C03633=1108.269,417.055,404.541,-178.654,16.489,151.227
C03634=1108.274,417.302,404.502,-178.652,16.496,151.228
C03635=1108.279,417.549,404.464,-178.650,16.503,151.230
C03636=1108.285,417.796,404.425,-178.649,16.510,151.231
C03637=1108.291,418.042,404.386,-178.647,16.517,151.232
C03638=1108.297,418.289,404.346,-178.645,16.524,151.234
C03639=1108.302,418.536,404.307,-178.644,16.531,151.235
C03640=1108.307,418.783,404.267,-178.642,16.538,151.237
C03641=1108.313,419.030,404.228,-178.640,16.545,151.238
C03642=1108.319,419.276,404.189,-178.639,16.553,151.240
C03643=1108.325,419.523,404.149,-178.638,16.560,151.241
C03644=1108.330,419.770,404.110,-178.636,16.567,151.243
C03645=1108.336,420.017,404.071,-178.634,16.574,151.244
C03646=1108.342,420.264,404.033,-178.632,16.582,151.246
C03647=1108.347,420.510,403.992,-178.631,16.589,151.247
C03648=1108.353,420.757,403.953,-178.629,16.596,151.249
C03649=1108.358,421.004,403.914,-178.627,16.603,151.250
C03650=1108.364,421.251,403.874,-178.626,16.611,151.252
C03651=1108.370,421.497,403.835,-178.625,16.618,151.254
C03652=1108.375,421.745,403.795,-178.623,16.625,151.255
C03653=1108.381,421.991,403.756,-178.621,16.633,151.257
C03654=1108.387,422.238,403.717,-178.619,16.640,151.258
C03655=1108.392,422.485,403.678,-178.618,16.648,151.260
C03656=1108.398,422.732,403.638,-178.616,16.655,151.261
C03657=1108.403,422.978,403.598,-178.615,16.663,151.263
C03658=1108.409,423.225,403.558,-178.614,16.670,151.265
C03659=1108.414,423.443,403.524,-178.612,16.678,151.266
C03660=1108.419,423.661,403.489,-178.611,16.684,151.268
C03661=1108.424,423.879,403.454,-178.610,16.691,151.269
C03662=1108.429,424.099,403.418,-178.608,16.698,151.271
C03663=1108.434,424.317,403.383,-178.607,16.704,151.272
C03664=1108.439,424.535,403.348,-178.606,16.712,151.274
C03665=1108.443,424.753,403.313,-178.604,16.718,151.275
C03666=1108.449,424.972,403.278,-178.603,16.725,151.277
C03667=1108.454,425.218,403.238,-178.602,16.733,151.278
C03668=1108.460,425.465,403.198,-178.600,16.741,151.280
C03669=1108.465,425.712,403.158,-178.599,16.749,151.282
C03670=1108.471,425.959,403.119,-178.598,16.757,151.283
C03671=1108.477,426.205,403.079,-178.596,16.764,151.285
C03672=1108.482,426.452,403.039,-178.595,16.773,151.287
C03673=1108.488,426.698,402.999,-178.593,16.781,151.289
C03674=1108.493,426.945,402.959,-178.592,16.789,151.290
C03675=1108.500,427.192,402.919,-178.591,16.797,151.292
C03676=1108.504,427.439,402.879,-178.589,16.805,151.294
C03677=1108.511,427.685,402.839,-178.588,16.813,151.296
C03678=1108.515,427.932,402.800,-178.587,16.821,151.298
C03679=1108.522,428.178,402.760,-178.585,16.829,151.299
C03680=1108.527,428.426,402.719,-178.584,16.837,151.301
C03681=1108.533,428.672,402.680,-178.583,16.845,151.303
C03682=1108.539,428.918,402.639,-178.582,16.854,151.305
C03683=1108.544,429.165,402.600,-178.580,16.862,151.307
C03684=1108.550,429.412,402.559,-178.579,16.870,151.309
C03685=1108.556,429.659,402.520,-178.578,16.879,151.311
C03686=1108.561,429.905,402.479,-178.577,16.887,151.312
C03687=1108.566,430.152,402.439,-178.575,16.896,151.314
C03688=1108.572,430.398,402.399,-178.574,16.904,151.316
C03689=1108.578,430.645,402.359,-178.573,16.913,151.318
C03690=1108.584,430.892,402.319,-178.572,16.921,151.320
C03691=1108.589,431.138,402.278,-178.571,16.930,151.322
C03692=1108.595,431.384,402.238,-178.570,16.938,151.324
C03693=1108.601,431.632,402.198,-178.568,16.946,151.326
C03694=1108.606,431.878,402.158,-178.567,16.956,151.328
C03695=1108.611,432.125,402.117,-178.566,16.964,151.330
C03696=1108.617,432.371,402.076,-178.565,16.973,151.332
C03697=1108.623,432.617,402.036,-178.564,16.981,151.334
C03698=1108.628,432.864,401.996,-178.563,16.990,151.336
C03699=1108.634,433.111,401.956,-178.561,16.999,151.338
C03700=1108.640,433.357,401.916,-178.560,17.008,151.340
C03701=1108.645,433.604,401.875,-178.560,17.017,151.342
C03702=1108.651,433.851,401.834,-178.559,17.025,151.344
C03703=1108.656,434.097,401.794,-178.558,17.034,151.346
C03704=1108.662,434.344,401.753,-178.556,17.044,151.348
C03705=1108.667,434.591,401.713,-178.556,17.052,151.351
C03706=1108.673,434.837,401.673,-178.555,17.061,151.353
C03707=1108.679,435.083,401.632,-178.553,17.071,151.355
C03708=1108.684,435.330,401.591,-178.553,17.080,151.357
C03709=1108.689,435.576,401.551,-178.552,17.089,151.359
C03710=1108.695,435.823,401.510,-178.551,17.098,151.361
C03711=1108.701,436.069,401.469,-178.550,17.107,151.364
C03712=1108.706,436.315,401.428,-178.549,17.117,151.366
C03713=1108.712,436.562,401.388,-178.549,17.126,151.368
C03714=1108.717,436.809,401.347,-178.547,17.135,151.370
C03715=1108.723,437.037,401.310,-178.546,17.144,151.372
C03716=1108.727,437.265,401.272,-178.545,17.153,151.374
C03717=1108.733,437.493,401.234,-178.545,17.161,151.376
C03718=1108.738,437.721,401.196,-178.545,17.170,151.379
C03719=1108.743,437.949,401.159,-178.544,17.179,151.381
C03720=1108.749,438.177,401.121,-178.543,17.188,151.383
C03721=1108.754,438.406,401.083,-178.542,17.196,151.385
C03722=1108.758,438.634,401.046,-178.541,17.205,151.387
C03723=1108.764,438.880,401.004,-178.541,17.215,151.389
C03724=1108.770,439.127,400.963,-178.540,17.224,151.392
C03725=1108.776,439.373,400.922,-178.539,17.234,151.394
C03726=1108.782,439.620,400.881,-178.538,17.244,151.396
C03727=1108.787,439.866,400.841,-178.538,17.254,151.399
C03728=1108.793,440.112,400.799,-178.537,17.264,151.401
C03729=1108.798,440.359,400.759,-178.536,17.273,151.403
C03730=1108.804,440.606,400.718,-178.536,17.283,151.406
C03731=1108.810,440.852,400.676,-178.535,17.293,151.408
C03732=1108.815,441.098,400.636,-178.535,17.303,151.411
C03733=1108.821,441.345,400.595,-178.534,17.313,151.413
C03734=1108.826,441.591,400.554,-178.534,17.323,151.416
C03735=1108.832,441.838,400.512,-178.533,17.333,151.418
C03736=1108.838,442.084,400.470,-178.532,17.343,151.420
C03737=1108.843,442.330,400.430,-178.532,17.353,151.423
C03738=1108.849,442.576,400.389,-178.531,17.364,151.426
C03739=1108.854,442.823,400.348,-178.530,17.374,151.428
C03740=1108.860,443.069,400.306,-178.530,17.384,151.431
C03741=1108.865,443.317,400.265,-178.530,17.394,151.433
C03742=1108.871,443.563,400.224,-178.529,17.405,151.436
C03743=1108.876,443.808,400.182,-178.529,17.415,151.438
C03744=1108.881,444.055,400.141,-178.529,17.425,151.441
C03745=1108.887,444.302,400.100,-178.529,17.435,151.444
C03746=1108.893,444.548,400.058,-178.529,17.445,151.446
C03747=1108.899,444.795,400.017,-178.530,17.456,151.449
C03748=1108.904,445.041,399.975,-178.530,17.466,151.452
C03749=1108.910,445.287,399.934,-178.530,17.477,151.454
C03750=1108.916,445.534,399.892,-178.531,17.486,151.457
C03751=1108.921,445.781,399.851,-178.531,17.497,151.460
C03752=1108.926,446.026,399.810,-178.532,17.506,151.463
C03753=1108.932,446.272,399.769,-178.533,17.517,151.465
C03754=1108.937,446.519,399.727,-178.534,17.527,151.468
C03755=1108.943,446.766,399.686,-178.535,17.537,151.471
C03756=1108.948,447.012,399.644,-178.537,17.547,151.474
C03757=1108.954,447.259,399.602,-178.538,17.557,151.477
C03758=1108.959,447.505,399.560,-178.539,17.567,151.480
C03759=1108.965,447.751,399.519,-178.540,17.577,151.482
C03760=1108.970,447.998,399.477,-178.541,17.587,151.485
C03761=1108.976,448.245,399.436,-178.544,17.597,151.488
C03762=1108.981,448.491,399.394,-178.545,17.608,151.491
C03763=1108.987,448.737,399.352,-178.547,17.617,151.494
C03764=1108.993,448.983,399.311,-178.549,17.628,151.497
C03765=1108.998,449.230,399.269,-178.551,17.637,151.500
C03766=1109.004,449.476,399.228,-178.553,17.647,151.503
C03767=1109.010,449.723,399.185,-178.555,17.658,151.506
C03768=1109.016,449.969,399.144,-178.557,17.667,151.509
C03769=1109.020,450.216,399.103,-178.559,17.677,151.512
C03770=1109.026,450.462,399.061,-178.561,17.687,151.515
C03771=1108.617,450.455,398.951,-178.646,17.920,151.591
C03772=1108.612,450.209,398.993,-178.644,17.910,151.588
C03773=1108.606,449.963,399.035,-178.642,17.900,151.585
C03774=1108.600,449.716,399.077,-178.640,17.890,151.582
C03775=1108.594,449.470,399.118,-178.638,17.880,151.579
C03776=1108.589,449.223,399.160,-178.635,17.870,151.576
C03777=1108.583,448.977,399.202,-178.634,17.859,151.573
C03778=1108.578,448.731,399.244,-178.632,17.850,151.570
C03779=1108.572,448.484,399.285,-178.631,17.839,151.568
C03780=1108.567,448.238,399.327,-178.628,17.830,151.565
C03781=1108.561,447.992,399.369,-178.627,17.819,151.562
C03782=1108.556,447.745,399.411,-178.626,17.809,151.559
C03783=1108.550,447.498,399.452,-178.624,17.799,151.556
C03784=1108.545,447.252,399.494,-178.622,17.789,151.553
C03785=1108.539,447.006,399.535,-178.621,17.779,151.550
C03786=1108.534,446.759,399.577,-178.620,17.769,151.547
C03787=1108.528,446.513,399.619,-178.620,17.758,151.544
C03788=1108.523,446.266,399.661,-178.618,17.748,151.542
C03789=1108.517,446.020,399.702,-178.617,17.738,151.539
C03790=1108.511,445.773,399.743,-178.617,17.727,151.536
C03791=1108.506,445.528,399.785,-178.616,17.717,151.533
C03792=1108.500,445.281,399.826,-178.616,17.707,151.530
C03793=1108.495,445.035,399.867,-178.615,17.696,151.528
C03794=1108.489,444.789,399.910,-178.615,17.687,151.525
C03795=1108.484,444.542,399.950,-178.614,17.676,151.522
C03796=1108.478,444.296,399.992,-178.614,17.666,151.520
C03797=1108.472,444.049,400.034,-178.614,17.656,151.517
C03798=1108.467,443.803,400.075,-178.615,17.645,151.515
C03799=1108.461,443.556,400.116,-178.615,17.635,151.512
C03800=1108.456,443.310,400.158,-178.616,17.624,151.509
C03801=1108.450,443.064,400.199,-178.616,17.614,151.507
C03802=1108.445,442.817,400.240,-178.617,17.603,151.504
C03803=1108.439,442.571,400.281,-178.617,17.593,151.502
C03804=1108.434,442.325,400.323,-178.618,17.583,151.499
C03805=1108.428,442.078,400.364,-178.618,17.573,151.497
C03806=1108.422,441.832,400.406,-178.619,17.563,151.494
C03807=1108.417,441.585,400.446,-178.620,17.552,151.492
C03808=1108.411,441.339,400.487,-178.620,17.542,151.489
C03809=1108.405,441.092,400.528,-178.621,17.532,151.487
C03810=1108.400,440.846,400.570,-178.621,17.522,151.484
C03811=1108.394,440.600,400.612,-178.622,17.511,151.482
C03812=1108.389,440.353,400.652,-178.623,17.502,151.479
C03813=1108.383,440.106,400.693,-178.624,17.492,151.477
C03814=1108.378,439.861,400.734,-178.624,17.482,151.475
C03815=1108.372,439.614,400.775,-178.625,17.472,151.472
C03816=1108.366,439.368,400.816,-178.626,17.462,151.470
C03817=1108.360,439.121,400.857,-178.626,17.453,151.467
C03818=1108.354,438.874,400.899,-178.628,17.443,151.465
C03819=1108.349,438.628,400.939,-178.628,17.433,151.463
C03820=1108.344,438.401,400.977,-178.629,17.425,151.461
C03821=1108.339,438.174,401.014,-178.630,17.416,151.459
C03822=1108.333,437.948,401.052,-178.631,17.407,151.456
C03823=1108.328,437.721,401.090,-178.631,17.398,151.454
C03824=1108.323,437.494,401.127,-178.632,17.389,151.452
C03825=1108.318,437.267,401.165,-178.633,17.380,151.450
C03826=1108.313,437.041,401.202,-178.634,17.371,151.448
C03827=1108.308,436.815,401.240,-178.634,17.363,151.446
C03828=1108.302,436.568,401.281,-178.636,17.354,151.444
C03829=1108.297,436.321,401.321,-178.636,17.344,151.442
C03830=1108.291,436.074,401.362,-178.637,17.335,151.439
C03831=1108.286,435.828,401.403,-178.639,17.326,151.437
C03832=1108.280,435.581,401.443,-178.639,17.316,151.435
C03833=1108.274,435.335,401.484,-178.640,17.308,151.433
C03834=1108.269,435.089,401.524,-178.641,17.298,151.431
C03835=1108.263,434.843,401.565,-178.642,17.289,151.428
C03836=1108.257,434.596,401.606,-178.643,17.280,151.426
C03837=1108.252,434.350,401.646,-178.644,17.270,151.424
C03838=1108.247,434.103,401.687,-178.645,17.261,151.422
C03839=1108.241,433.856,401.728,-178.646,17.252,151.420
C03840=1108.236,433.610,401.768,-178.648,17.243,151.418
C03841=1108.230,433.363,401.808,-178.649,17.234,151.416
C03842=1108.224,433.116,401.849,-178.650,17.225,151.414
C03843=1108.218,432.870,401.890,-178.650,17.217,151.412
C03844=1108.213,432.623,401.930,-178.651,17.208,151.410
C03845=1108.207,432.377,401.970,-178.653,17.198,151.408
C03846=1108.201,432.130,402.011,-178.654,17.190,151.406
C03847=1108.196,431.883,402.051,-178.655,17.181,151.404
C03848=1108.190,431.637,402.091,-178.656,17.173,151.402
C03849=1108.184,431.390,402.132,-178.657,17.164,151.400
C03850=1108.179,431.144,402.172,-178.659,17.155,151.398
C03851=1108.173,430.897,402.212,-178.660,17.146,151.396
C03852=1108.167,430.651,402.253,-178.661,17.138,151.394
C03853=1108.163,430.404,402.293,-178.662,17.129,151.392
C03854=1108.156,430.157,402.333,-178.663,17.121,151.390
C03855=1108.151,429.911,402.373,-178.665,17.113,151.388
C03856=1108.146,429.664,402.413,-178.667,17.104,151.386
C03857=1108.139,429.417,402.453,-178.668,17.095,151.384
C03858=1108.134,429.171,402.494,-178.669,17.087,151.382
C03859=1108.128,428.925,402.534,-178.670,17.078,151.380
C03860=1108.123,428.677,402.574,-178.671,17.070,151.378
C03861=1108.118,428.431,402.614,-178.673,17.062,151.377
C03862=1108.112,428.184,402.654,-178.674,17.054,151.375
C03863=1108.106,427.937,402.694,-178.675,17.046,151.373
C03864=1108.100,427.691,402.734,-178.677,17.037,151.371
C03865=1108.095,427.444,402.774,-178.678,17.029,151.369
C03866=1108.089,427.198,402.814,-178.679,17.021,151.367
C03867=1108.083,426.951,402.853,-178.681,17.013,151.366
C03868=1108.077,426.704,402.894,-178.682,17.005,151.364
C03869=1108.072,426.458,402.933,-178.684,16.997,151.362
C03870=1108.066,426.211,402.974,-178.685,16.989,151.360
C03871=1108.061,425.964,403.013,-178.686,16.981,151.359
C03872=1108.055,425.718,403.054,-178.688,16.973,151.357
C03873=1108.050,425.471,403.093,-178.689,16.965,151.355
C03874=1108.044,425.224,403.133,-178.691,16.957,151.353
C03875=1108.039,424.978,403.173,-178.692,16.949,151.352
C03876=1108.033,424.759,403.207,-178.693,16.942,151.350
C03877=1108.029,424.540,403.243,-178.695,16.935,151.349
C03878=1108.023,424.322,403.279,-178.696,16.928,151.347
C03879=1108.019,424.103,403.313,-178.697,16.921,151.346
C03880=1108.013,423.885,403.348,-178.699,16.914,151.344
C03881=1108.009,423.666,403.384,-178.700,16.907,151.343
C03882=1108.004,423.448,403.419,-178.702,16.901,151.341
C03883=1107.999,423.230,403.454,-178.703,16.894,151.340
C03884=1107.993,422.983,403.494,-178.704,16.886,151.338
C03885=1107.988,422.736,403.533,-178.706,16.878,151.336
C03886=1107.982,422.489,403.573,-178.708,16.871,151.335
C03887=1107.976,422.243,403.613,-178.709,16.863,151.333
C03888=1107.970,421.996,403.652,-178.711,16.855,151.332
C03889=1107.965,421.750,403.691,-178.712,16.848,151.330
C03890=1107.959,421.502,403.731,-178.714,16.841,151.329
C03891=1107.954,421.256,403.770,-178.715,16.833,151.327
C03892=1107.948,421.009,403.810,-178.717,16.826,151.325
C03893=1107.942,420.762,403.849,-178.719,16.818,151.324
C03894=1107.936,420.515,403.888,-178.720,16.811,151.322
C03895=1107.931,420.268,403.928,-178.722,16.804,151.321
C03896=1107.925,420.021,403.967,-178.724,16.796,151.319
C03897=1107.920,419.775,404.007,-178.725,16.789,151.318
C03898=1107.914,419.528,404.046,-178.727,16.782,151.316
C03899=1107.908,419.282,404.085,-178.728,16.775,151.315
C03900=1107.902,419.034,404.124,-178.730,16.767,151.313
C03901=1107.898,418.787,404.164,-178.732,16.760,151.312
C03902=1107.891,418.540,404.203,-178.734,16.753,151.310
C03903=1107.886,418.294,404.242,-178.735,16.746,151.309
C03904=1107.881,418.047,404.281,-178.737,16.738,151.307
C03905=1107.874,417.800,404.321,-178.739,16.731,151.306
C03906=1107.869,417.554,404.360,-178.740,16.725,151.304
C03907=1107.863,417.307,404.399,-178.742,16.717,151.303
C03908=1107.857,417.060,404.438,-178.744,16.710,151.302
C03909=1107.853,416.813,404.477,-178.746,16.703,151.300
C03910=1107.847,416.566,404.517,-178.747,16.696,151.299
C03911=1107.841,416.320,404.555,-178.749,16.689,151.297
C03912=1107.835,416.072,404.595,-178.751,16.683,151.296
C03913=1107.829,415.826,404.634,-178.753,16.676,151.294
C03914=1107.823,415.578,404.672,-178.755,16.669,151.293
C03915=1107.818,415.332,404.712,-178.756,16.662,151.292
C03916=1107.812,415.085,404.751,-178.758,16.655,151.290
C03917=1107.807,414.838,404.789,-178.760,16.649,151.289
C03918=1107.801,414.591,404.828,-178.762,16.642,151.288
C03919=1107.795,414.344,404.868,-178.764,16.635,151.286
C03920=1107.790,414.097,404.906,-178.765,16.628,151.285
C03921=1107.785,413.851,404.945,-178.768,16.621,151.284
C03922=1107.778,413.604,404.984,-178.769,16.615,151.282
C03923=1107.773,413.357,405.022,-178.771,16.608,151.281
C03924=1107.767,413.110,405.061,-178.773,16.602,151.280
C03925=1107.761,412.863,405.100,-178.775,16.595,151.279
C03926=1107.756,412.616,405.139,-178.776,16.589,151.277
C03927=1107.751,412.369,405.178,-178.779,16.582,151.276
C03928=1107.745,412.122,405.217,-178.780,16.576,151.275
C03929=1107.739,411.875,405.255,-178.782,16.569,151.273
C03930=1107.733,411.629,405.294,-178.784,16.563,151.272
C03931=1107.727,411.381,405.333,-178.786,16.556,151.271
C03932=1107.723,411.169,405.366,-178.788,16.550,151.270
C03933=1107.717,410.957,405.399,-178.789,16.545,151.269
C03934=1107.713,410.746,405.432,-178.791,16.539,151.268
C03935=1107.708,410.534,405.465,-178.793,16.534,151.267
C03936=1107.703,410.322,405.498,-178.794,16.529,151.266
C03937=1107.699,410.109,405.531,-178.796,16.523,151.265
C03938=1107.694,409.897,405.564,-178.798,16.517,151.264
C03939=1107.689,409.686,405.598,-178.799,16.512,151.263
C03940=1107.683,409.439,405.636,-178.802,16.506,151.261
C03941=1107.677,409.191,405.675,-178.803,16.500,151.260
C03942=1107.672,408.945,405.714,-178.805,16.494,151.259
C03943=1107.667,408.698,405.752,-178.807,16.487,151.258
C03944=1107.661,408.451,405.790,-178.809,16.481,151.257
C03945=1107.656,408.204,405.828,-178.811,16.474,151.256
C03946=1107.650,407.956,405.867,-178.813,16.468,151.254
C03947=1107.644,407.710,405.905,-178.815,16.463,151.253
C03948=1107.639,407.463,405.944,-178.817,16.456,151.252
C03949=1107.633,407.216,405.982,-178.819,16.450,151.251
C03950=1107.627,406.968,406.020,-178.821,16.444,151.250
C03951=1107.622,406.721,406.059,-178.823,16.438,151.249
C03952=1107.616,406.475,406.098,-178.825,16.432,151.248
C03953=1107.610,406.228,406.135,-178.827,16.426,151.247
C03954=1107.605,405.981,406.174,-178.829,16.420,151.245
C03955=1107.599,405.734,406.212,-178.831,16.414,151.244
C03956=1107.594,405.487,406.250,-178.833,16.408,151.243
C03957=1107.588,405.240,406.288,-178.835,16.402,151.242
C03958=1107.582,404.993,406.326,-178.838,16.396,151.241
C03959=1107.577,404.746,406.364,-178.839,16.391,151.240
C03960=1107.571,404.498,406.403,-178.841,16.385,151.239
C03961=1107.565,404.252,406.441,-178.843,16.379,151.238
C03962=1107.560,404.005,406.479,-178.846,16.373,151.237
C03963=1107.554,403.758,406.517,-178.848,16.367,151.236
C03964=1107.549,403.511,406.555,-178.850,16.362,151.235
C03965=1107.542,403.263,406.593,-178.852,16.356,151.234
C03966=1107.536,403.017,406.631,-178.854,16.351,151.233
C03967=1107.531,402.769,406.669,-178.856,16.345,151.232
C03968=1107.525,402.523,406.707,-178.859,16.339,151.231
C03969=1107.520,402.275,406.745,-178.860,16.333,151.230
C03970=1107.514,402.028,406.782,-178.863,16.328,151.229
C03971=1107.509,401.782,406.820,-178.865,16.322,151.228
C03972=1107.503,401.535,406.858,-178.867,16.317,151.227
C03973=1107.497,401.287,406.897,-178.869,16.311,151.226
C03974=1107.492,401.040,406.935,-178.871,16.305,151.225
C03975=1107.486,400.793,406.972,-178.874,16.300,151.224
C03976=1107.480,400.546,407.010,-178.876,16.294,151.223
C03977=1107.475,400.299,407.048,-178.878,16.289,151.223
C03978=1107.469,400.052,407.086,-178.880,16.284,151.222
C03979=1107.464,399.805,407.123,-178.882,16.278,151.221
C03980=1107.458,399.558,407.161,-178.884,16.273,151.220
C03981=1107.452,399.311,407.199,-178.886,16.267,151.219
C03982=1107.447,399.064,407.236,-178.888,16.262,151.218
C03983=1107.441,398.817,407.274,-178.890,16.257,151.217
C03984=1107.435,398.570,407.312,-178.893,16.251,151.216
C03985=1107.430,398.322,407.349,-178.895,16.246,151.215
C03986=1107.424,398.076,407.387,-178.897,16.241,151.214
C03987=1107.418,397.829,407.425,-178.899,16.235,151.214
C03988=1107.414,397.616,407.457,-178.902,16.231,151.213
C03989=1107.408,397.404,407.489,-178.903,16.226,151.212
C03990=1107.404,397.192,407.522,-178.905,16.222,151.211
C03991=1107.398,396.979,407.553,-178.907,16.217,151.211
C03992=1107.394,396.768,407.586,-178.909,16.213,151.210
C03993=1107.389,396.555,407.618,-178.911,16.208,151.209
C03994=1107.384,396.343,407.650,-178.913,16.204,151.209
C03995=1107.380,396.131,407.683,-178.915,16.199,151.208
C03996=1107.374,395.884,407.720,-178.917,16.194,151.207
C03997=1107.368,395.637,407.757,-178.920,16.189,151.206
C03998=1107.363,395.390,407.794,-178.922,16.184,151.205
C03999=1107.357,395.143,407.832,-178.924,16.179,151.205
C04000=1107.351,394.896,407.869,-178.927,16.174,151.204
C04001=1107.346,394.648,407.906,-178.929,16.168,151.203
C04002=1107.340,394.401,407.944,-178.931,16.164,151.202
C04003=1107.334,394.154,407.981,-178.934,16.159,151.202
C04004=1107.328,393.907,408.019,-178.936,16.153,151.201
C04005=1107.323,393.660,408.056,-178.938,16.149,151.200
C04006=1107.317,393.413,408.093,-178.940,16.144,151.199
C04007=1107.311,393.166,408.131,-178.943,16.139,151.198
C04008=1107.306,392.919,408.168,-178.945,16.134,151.198
C04009=1107.300,392.671,408.205,-178.948,16.129,151.197
C04010=1107.294,392.424,408.242,-178.950,16.124,151.196
C04011=1107.289,392.178,408.279,-178.953,16.119,151.196
C04012=1107.283,391.930,408.316,-178.955,16.115,151.195
C04013=1107.278,391.683,408.353,-178.958,16.110,151.194
C04014=1107.272,391.436,408.390,-178.960,16.105,151.193
C04015=1107.266,391.189,408.427,-178.962,16.101,151.193
C04016=1107.260,390.942,408.464,-178.964,16.096,151.192
C04017=1107.254,390.695,408.501,-178.967,16.091,151.191
C04018=1107.249,390.447,408.538,-178.969,16.086,151.191
C04019=1107.243,390.200,408.576,-178.972,16.081,151.190
C04020=1107.238,389.954,408.613,-178.975,16.076,151.189
C04021=1107.232,389.707,408.649,-178.977,16.072,151.189
C04022=1107.226,389.459,408.686,-178.979,16.067,151.188
C04023=1107.220,389.212,408.723,-178.981,16.062,151.187
C04024=1107.215,388.965,408.760,-178.984,16.058,151.187
C04025=1107.208,388.718,408.797,-178.987,16.053,151.186
C04026=1107.203,388.471,408.834,-178.989,16.048,151.186
C04027=1107.198,388.224,408.871,-178.992,16.044,151.185
C04028=1107.192,387.976,408.908,-178.994,16.040,151.184
C04029=1107.186,387.729,408.944,-178.996,16.035,151.184
C04030=1107.180,387.482,408.981,-178.999,16.030,151.183
C04031=1107.175,387.235,409.018,-179.002,16.025,151.182
C04032=1107.170,386.988,409.055,-179.004,16.021,151.182
C04033=1107.163,386.741,409.091,-179.007,16.016,151.181
C04034=1107.158,386.493,409.128,-179.009,16.012,151.181
C04035=1107.153,386.247,409.165,-179.012,16.008,151.180
C04036=1107.146,386.000,409.201,-179.014,16.003,151.179
C04037=1107.141,385.752,409.239,-179.017,15.998,151.179
C04038=1107.136,385.506,409.275,-179.019,15.994,151.178
C04039=1107.130,385.259,409.312,-179.022,15.990,151.178
C04040=1107.124,385.011,409.348,-179.024,15.985,151.177
C04041=1107.119,384.763,409.385,-179.027,15.980,151.176
C04042=1107.113,384.517,409.421,-179.029,15.977,151.176
C04043=1107.107,384.269,409.458,-179.032,15.972,151.175
C04044=1107.098,383.857,409.519,-179.036,15.965,151.175
C04045=1107.089,383.444,409.580,-179.041,15.957,151.174
C04046=1107.080,383.032,409.641,-179.045,15.950,151.173
C04047=1107.070,382.620,409.702,-179.049,15.943,151.172
C04048=1107.064,382.373,409.737,-179.052,15.939,151.171
C04049=1107.059,382.126,409.774,-179.055,15.935,151.171
C04050=1107.052,381.879,409.811,-179.057,15.930,151.170
C04051=1107.048,381.631,409.847,-179.060,15.926,151.170
C04052=1107.041,381.384,409.883,-179.063,15.922,151.169
C04053=1107.036,381.136,409.920,-179.065,15.918,151.169
C04054=1107.030,380.889,409.956,-179.068,15.913,151.168
C04055=1107.024,380.643,409.992,-179.070,15.910,151.168
C04056=1107.019,380.395,410.028,-179.073,15.905,151.167
C04057=1107.012,380.148,410.065,-179.076,15.902,151.167
C04058=1107.008,379.901,410.101,-179.078,15.897,151.167
C04059=1107.001,379.653,410.137,-179.081,15.893,151.166
C04060=1106.996,379.407,410.173,-179.083,15.889,151.166
C04061=1106.990,379.159,410.210,-179.087,15.885,151.165
C04062=1106.984,378.911,410.245,-179.089,15.881,151.165
C04063=1106.978,378.665,410.281,-179.092,15.877,151.164
C04064=1106.973,378.417,410.318,-179.095,15.873,151.164
C04065=1106.967,378.169,410.353,-179.098,15.868,151.163
C04066=1106.962,377.923,410.390,-179.100,15.865,151.163
C04067=1106.956,377.675,410.426,-179.103,15.861,151.163
C04068=1106.950,377.429,410.462,-179.105,15.857,151.162
C04069=1106.945,377.181,410.498,-179.108,15.853,151.162
C04070=1106.940,376.934,410.534,-179.111,15.849,151.161
C04071=1106.933,376.687,410.570,-179.113,15.845,151.161
C04072=1106.928,376.439,410.606,-179.117,15.841,151.161
C04073=1106.923,376.192,410.642,-179.119,15.838,151.160
C04074=1106.916,375.945,410.678,-179.122,15.833,151.160
C04075=1106.911,375.698,410.714,-179.124,15.830,151.159
C04076=1106.906,375.450,410.750,-179.127,15.825,151.159
C04077=1106.900,375.203,410.785,-179.130,15.821,151.159
C04078=1106.894,374.955,410.821,-179.132,15.818,151.158
C04079=1106.888,374.709,410.857,-179.136,15.814,151.158
C04080=1106.883,374.461,410.893,-179.138,15.810,151.158
C04081=1106.878,374.214,410.929,-179.141,15.806,151.157
C04082=1106.872,373.966,410.965,-179.144,15.803,151.157
C04083=1106.866,373.718,411.000,-179.147,15.799,151.157
C04084=1106.860,373.472,411.036,-179.149,15.795,151.156
C04085=1106.854,373.224,411.072,-179.152,15.792,151.156
C04086=1106.848,372.977,411.107,-179.155,15.788,151.156
C04087=1106.842,372.730,411.143,-179.158,15.784,151.155
C04088=1106.838,372.483,411.179,-179.161,15.781,151.155
C04089=1106.832,372.235,411.215,-179.164,15.777,151.155
C04090=1106.826,371.988,411.250,-179.166,15.773,151.154
C04091=1106.820,371.740,411.286,-179.169,15.769,151.154
C04092=1106.815,371.493,411.321,-179.172,15.766,151.154
C04093=1106.809,371.246,411.357,-179.175,15.762,151.154
C04094=1106.803,370.999,411.392,-179.177,15.759,151.153
C04095=1106.797,370.751,411.428,-179.181,15.755,151.153
C04096=1106.788,370.365,411.483,-179.185,15.749,151.152
C04097=1106.779,369.980,411.539,-179.190,15.744,151.152
C04098=1106.770,369.594,411.594,-179.194,15.738,151.152
C04099=1106.762,369.208,411.649,-179.199,15.733,151.151
C04100=1106.757,368.961,411.685,-179.201,15.729,151.151
C04101=1106.751,368.714,411.720,-179.204,15.725,151.151
C04102=1106.746,368.467,411.756,-179.207,15.722,151.150
C04103=1106.739,368.219,411.790,-179.209,15.719,151.150
C04104=1106.734,367.972,411.826,-179.213,15.715,151.150
C04105=1106.728,367.725,411.861,-179.215,15.712,151.150
C04106=1106.722,367.477,411.897,-179.219,15.708,151.149
C04107=1106.717,367.229,411.931,-179.221,15.705,151.149
C04108=1106.711,366.982,411.967,-179.225,15.701,151.149
C04109=1106.706,366.735,412.002,-179.227,15.698,151.149
C04110=1106.700,366.488,412.038,-179.230,15.695,151.148
C04111=1106.694,366.239,412.073,-179.233,15.691,151.148
C04112=1106.689,365.993,412.108,-179.236,15.688,151.148
C04113=1106.683,365.744,412.143,-179.239,15.684,151.148
C04114=1106.678,365.497,412.179,-179.242,15.681,151.148
C04115=1106.672,365.251,412.213,-179.244,15.678,151.147
C04116=1106.666,365.002,412.248,-179.248,15.674,151.147
C04117=1106.661,364.755,412.284,-179.251,15.671,151.147
C04118=1106.655,364.508,412.319,-179.253,15.668,151.147
C04119=1106.649,364.260,412.354,-179.257,15.664,151.147
C04120=1106.643,364.013,412.389,-179.259,15.661,151.146
C04121=1106.637,363.765,412.424,-179.263,15.658,151.146
C04122=1106.632,363.518,412.459,-179.266,15.655,151.146
C04123=1106.627,363.271,412.494,-179.268,15.652,151.146
C04124=1106.620,363.023,412.529,-179.272,15.648,151.146
C04125=1106.615,362.776,412.564,-179.275,15.645,151.146
C04126=1106.610,362.529,412.599,-179.277,15.642,151.146
C04127=1106.603,362.281,412.633,-179.281,15.638,151.145
C04128=1106.598,362.033,412.668,-179.284,15.635,151.145
C04129=1106.593,361.786,412.703,-179.286,15.632,151.145
C04130=1106.586,361.538,412.738,-179.290,15.629,151.145
C04131=1106.581,361.291,412.773,-179.292,15.626,151.145
C04132=1106.576,361.043,412.808,-179.295,15.623,151.145
C04133=1106.569,360.795,412.842,-179.299,15.619,151.145
C04134=1106.564,360.549,412.878,-179.301,15.616,151.144
C04135=1106.559,360.301,412.912,-179.304,15.613,151.144
C04136=1106.553,360.054,412.946,-179.308,15.610,151.144
C04137=1106.547,359.806,412.982,-179.311,15.607,151.144
C04138=1106.542,359.558,413.017,-179.313,15.604,151.144
C04139=1106.536,359.311,413.051,-179.316,15.601,151.144
C04140=1106.530,359.063,413.086,-179.320,15.598,151.144
C04141=1106.524,358.816,413.121,-179.323,15.595,151.144
C04142=1106.519,358.569,413.155,-179.326,15.592,151.144
C04143=1106.512,358.321,413.190,-179.329,15.588,151.143
C04144=1106.507,358.073,413.224,-179.332,15.586,151.143
C04145=1106.501,357.826,413.258,-179.335,15.583,151.143
C04146=1106.496,357.579,413.294,-179.338,15.580,151.143
C04147=1106.489,357.331,413.328,-179.341,15.577,151.143
C04148=1106.481,356.960,413.380,-179.346,15.572,151.143
C04149=1106.472,356.589,413.432,-179.350,15.568,151.143
C04150=1106.464,356.218,413.483,-179.355,15.563,151.143
C04151=1106.457,355.847,413.535,-179.359,15.559,151.143
C04152=1106.450,355.599,413.569,-179.362,15.557,151.143
C04153=1106.444,355.352,413.603,-179.366,15.553,151.143
C04154=1106.439,355.105,413.638,-179.369,15.550,151.143
C04155=1106.433,354.857,413.672,-179.372,15.548,151.143
C04156=1106.428,354.610,413.706,-179.375,15.545,151.143
C04157=1106.422,354.362,413.741,-179.378,15.542,151.143
C04158=1106.417,354.114,413.776,-179.382,15.539,151.143
C04159=1106.411,353.867,413.810,-179.385,15.536,151.143
C04160=1106.405,353.620,413.844,-179.388,15.534,151.142
C04161=1106.400,353.372,413.878,-179.390,15.531,151.142
C04162=1106.394,353.125,413.912,-179.393,15.528,151.142
C04163=1106.388,352.877,413.947,-179.397,15.525,151.142
C04164=1106.382,352.629,413.981,-179.400,15.522,151.142
C04165=1106.377,352.381,414.015,-179.403,15.519,151.142
C04166=1106.371,352.134,414.049,-179.406,15.517,151.142
C04167=1106.366,351.886,414.083,-179.409,15.514,151.142
C04168=1106.360,351.639,414.117,-179.413,15.511,151.142
C04169=1106.354,351.391,414.152,-179.416,15.508,151.142
C04170=1106.348,351.143,414.185,-179.419,15.506,151.142
C04171=1106.343,350.896,414.220,-179.422,15.503,151.142
C04172=1106.337,350.648,414.254,-179.425,15.501,151.142
C04173=1106.331,350.401,414.288,-179.428,15.498,151.142
C04174=1106.326,350.153,414.321,-179.432,15.495,151.143
C04175=1106.320,349.905,414.356,-179.435,15.492,151.143
C04176=1106.315,349.658,414.390,-179.438,15.489,151.142
C04177=1106.308,349.410,414.424,-179.441,15.487,151.143
C04178=1106.303,349.162,414.458,-179.444,15.484,151.143
C04179=1106.297,348.915,414.492,-179.447,15.482,151.143
C04180=1106.292,348.667,414.526,-179.450,15.479,151.143
C04181=1106.286,348.420,414.560,-179.454,15.476,151.143
C04182=1106.280,348.172,414.593,-179.457,15.474,151.143
C04183=1106.275,347.924,414.627,-179.460,15.471,151.143
C04184=1106.269,347.677,414.661,-179.464,15.469,151.143
C04185=1106.263,347.429,414.695,-179.467,15.466,151.143
C04186=1106.257,347.182,414.729,-179.470,15.464,151.143
C04187=1106.253,346.934,414.763,-179.473,15.461,151.143
C04188=1106.247,346.686,414.797,-179.476,15.459,151.143
C04189=1106.241,346.438,414.830,-179.480,15.455,151.143
C04190=1106.235,346.191,414.864,-179.483,15.453,151.143
C04191=1106.230,345.943,414.897,-179.486,15.451,151.143
C04192=1106.224,345.696,414.931,-179.489,15.448,151.143
C04193=1106.218,345.448,414.965,-179.492,15.446,151.144
C04194=1106.213,345.200,414.998,-179.496,15.443,151.144
C04195=1106.206,344.952,415.033,-179.499,15.441,151.144
C04196=1106.201,344.704,415.066,-179.502,15.438,151.144
C04197=1106.195,344.457,415.100,-179.505,15.436,151.144
C04198=1106.189,344.209,415.133,-179.509,15.434,151.144
C04199=1106.184,343.961,415.167,-179.511,15.431,151.144
C04200=1106.176,343.593,415.216,-179.517,15.428,151.144
C04201=1106.167,343.224,415.266,-179.521,15.424,151.144
C04202=1106.158,342.856,415.316,-179.526,15.420,151.145
C04203=1106.150,342.487,415.366,-179.531,15.417,151.145
C04204=1106.144,342.239,415.399,-179.535,15.414,151.145
C04205=1106.139,341.991,415.433,-179.538,15.411,151.145
C04206=1106.133,341.744,415.467,-179.541,15.409,151.145
C04207=1106.127,341.496,415.500,-179.545,15.407,151.145
C04208=1106.122,341.248,415.533,-179.548,15.404,151.145
C04209=1106.117,341.001,415.566,-179.551,15.402,151.146
C04210=1106.110,340.753,415.599,-179.554,15.400,151.146
C04211=1106.104,340.506,415.633,-179.558,15.398,151.146
C04212=1106.099,340.258,415.667,-179.561,15.395,151.146
C04213=1106.093,340.010,415.700,-179.564,15.393,151.146
C04214=1106.088,339.762,415.733,-179.568,15.391,151.146
C04215=1106.082,339.514,415.767,-179.571,15.388,151.146
C04216=1106.076,339.267,415.799,-179.574,15.386,151.147
C04217=1106.070,339.019,415.833,-179.577,15.384,151.147
C04218=1106.065,338.771,415.866,-179.581,15.381,151.147
C04219=1106.059,338.523,415.899,-179.584,15.379,151.147
C04220=1106.054,338.276,415.932,-179.587,15.377,151.147
C04221=1106.048,338.028,415.965,-179.591,15.375,151.147
C04222=1106.042,337.780,415.998,-179.594,15.373,151.148
C04223=1106.037,337.532,416.032,-179.597,15.370,151.148
C04224=1106.031,337.285,416.064,-179.601,15.368,151.148
C04225=1106.025,337.037,416.098,-179.604,15.366,151.148
C04226=1106.020,336.789,416.131,-179.607,15.364,151.148
C04227=1106.013,336.541,416.164,-179.611,15.361,151.148
C04228=1106.008,336.293,416.197,-179.614,15.360,151.149
C04229=1106.003,336.046,416.230,-179.617,15.358,151.149
C04230=1105.996,335.799,416.263,-179.620,15.356,151.149
C04231=1105.991,335.550,416.296,-179.623,15.353,151.149
C04232=1105.986,335.302,416.329,-179.627,15.351,151.150
C04233=1105.979,335.055,416.362,-179.630,15.349,151.150
C04234=1105.974,334.807,416.395,-179.634,15.347,151.150
C04235=1105.969,334.559,416.428,-179.637,15.345,151.150
C04236=1105.963,334.311,416.460,-179.640,15.342,151.150
C04237=1105.957,334.063,416.493,-179.644,15.341,151.151
C04238=1105.951,333.816,416.526,-179.647,15.338,151.151
C04239=1105.945,333.568,416.559,-179.651,15.336,151.151
C04240=1105.941,333.320,416.592,-179.654,15.334,151.151
C04241=1105.935,333.072,416.624,-179.657,15.332,151.151
C04242=1105.929,332.824,416.658,-179.661,15.330,151.152
C04243=1105.923,332.576,416.690,-179.664,15.328,151.152
C04244=1105.918,332.329,416.723,-179.667,15.326,151.152
C04245=1105.912,332.081,416.755,-179.670,15.324,151.152
C04246=1105.906,331.833,416.788,-179.674,15.322,151.153
C04247=1105.900,331.585,416.821,-179.678,15.320,151.153
C04248=1105.895,331.337,416.854,-179.681,15.318,151.153
C04249=1105.889,331.089,416.886,-179.684,15.316,151.153
C04250=1105.883,330.842,416.919,-179.688,15.314,151.154
C04251=1105.877,330.594,416.952,-179.691,15.312,151.154
C04252=1105.869,330.219,417.000,-179.696,15.310,151.154
C04253=1105.860,329.845,417.050,-179.701,15.307,151.155
C04254=1105.851,329.470,417.099,-179.706,15.303,151.155
C04255=1105.842,329.095,417.148,-179.712,15.301,151.156
C04256=1105.837,328.847,417.181,-179.715,15.299,151.156
C04257=1105.831,328.599,417.213,-179.719,15.297,151.156
C04258=1105.825,328.351,417.246,-179.722,15.295,151.156
C04259=1105.820,328.103,417.278,-179.725,15.293,151.157
C04260=1105.814,327.856,417.311,-179.729,15.291,151.157
C04261=1105.808,327.608,417.343,-179.732,15.289,151.157
C04262=1105.802,327.360,417.374,-179.736,15.288,151.158
C04263=1105.797,327.112,417.408,-179.740,15.286,151.158
C04264=1105.791,326.864,417.440,-179.742,15.284,151.158
C04265=1105.785,326.616,417.472,-179.746,15.282,151.158
C04266=1105.779,326.369,417.504,-179.749,15.280,151.159
C04267=1105.774,326.120,417.537,-179.753,15.278,151.159
C04268=1105.768,325.872,417.569,-179.756,15.276,151.159
C04269=1105.762,325.625,417.601,-179.760,15.274,151.160
C04270=1105.756,325.377,417.633,-179.763,15.273,151.160
C04271=1105.751,325.129,417.666,-179.766,15.271,151.160
C04272=1105.745,324.882,417.698,-179.770,15.269,151.161
C04273=1105.739,324.633,417.730,-179.774,15.268,151.161
C04274=1105.734,324.386,417.762,-179.777,15.266,151.161
C04275=1105.728,324.138,417.794,-179.780,15.264,151.162
C04276=1105.723,323.889,417.827,-179.783,15.262,151.162
C04277=1105.717,323.642,417.859,-179.787,15.260,151.162
C04278=1105.711,323.394,417.891,-179.791,15.258,151.162
C04279=1105.705,323.147,417.923,-179.794,15.256,151.163
C04280=1105.699,322.898,417.955,-179.797,15.255,151.163
C04281=1105.693,322.650,417.987,-179.801,15.254,151.164
C04282=1105.689,322.402,418.019,-179.805,15.252,151.164
C04283=1105.683,322.154,418.051,-179.808,15.250,151.164
C04284=1105.677,321.907,418.083,-179.811,15.249,151.164
C04285=1105.671,321.659,418.115,-179.815,15.247,151.165
C04286=1105.666,321.412,418.147,-179.818,15.245,151.165
C04287=1105.660,321.163,418.179,-179.822,15.243,151.165
C04288=1105.654,320.916,418.211,-179.825,15.241,151.166
C04289=1105.648,320.668,418.243,-179.828,15.240,151.166
C04290=1105.643,320.420,418.274,-179.832,15.238,151.166
C04291=1105.638,320.172,418.307,-179.835,15.236,151.167
C04292=1105.632,319.924,418.339,-179.839,15.234,151.167
C04293=1105.626,319.676,418.371,-179.842,15.233,151.167
C04294=1105.621,319.428,418.402,-179.846,15.231,151.168
C04295=1105.615,319.179,418.434,-179.849,15.229,151.168
C04296=1105.610,318.932,418.465,-179.853,15.228,151.169
C04297=1105.604,318.684,418.497,-179.856,15.226,151.169
C04298=1105.599,318.436,418.529,-179.860,15.224,151.169
C04299=1105.593,318.188,418.561,-179.863,15.223,151.169
C04300=1105.587,317.941,418.593,-179.867,15.221,151.170
C04301=1105.581,317.692,418.625,-179.870,15.220,151.170
C04302=1105.576,317.445,418.657,-179.873,15.218,151.171
C04303=1105.571,317.197,418.687,-179.877,15.216,151.171
C04304=1105.562,316.815,418.736,-179.883,15.214,151.172
C04305=1105.554,316.433,418.786,-179.887,15.211,151.172
C04306=1105.545,316.051,418.834,-179.893,15.209,151.173
C04307=1105.536,315.669,418.883,-179.899,15.206,151.173
C04308=1105.531,315.421,418.915,-179.902,15.204,151.174
C04309=1105.525,315.173,418.946,-179.905,15.203,151.174
C04310=1105.519,314.925,418.977,-179.909,15.202,151.174
C04311=1105.513,314.678,419.009,-179.913,15.200,151.175
C04312=1105.508,314.429,419.040,-179.916,15.199,151.175
C04313=1105.502,314.181,419.072,-179.920,15.197,151.176
C04314=1105.496,313.934,419.103,-179.924,15.196,151.176
C04315=1105.491,313.685,419.134,-179.926,15.195,151.177
C04316=1105.485,313.437,419.166,-179.930,15.193,151.177
C04317=1105.478,313.190,419.197,-179.934,15.191,151.177
C04318=1105.473,312.941,419.229,-179.937,15.190,151.178
C04319=1105.467,312.694,419.260,-179.941,15.189,151.178
C04320=1105.462,312.446,419.291,-179.945,15.187,151.179
C04321=1105.456,312.198,419.323,-179.948,15.186,151.179
C04322=1105.450,311.950,419.354,-179.951,15.184,151.179
C04323=1105.444,311.702,419.385,-179.955,15.183,151.180
C04324=1105.438,311.454,419.417,-179.959,15.182,151.180
C04325=1105.433,311.206,419.447,-179.962,15.180,151.181
C04326=1105.427,310.958,419.479,-179.966,15.179,151.181
C04327=1105.421,310.710,419.510,-179.969,15.178,151.182
C04328=1105.415,310.463,419.541,-179.973,15.176,151.182
C04329=1105.410,310.214,419.572,-179.977,15.174,151.183
C04330=1105.404,309.967,419.603,-179.980,15.174,151.183
C04331=1105.398,309.719,419.634,-179.984,15.172,151.183
C04332=1105.393,309.470,419.666,-179.988,15.170,151.184
C04333=1105.387,309.223,419.697,-179.991,15.169,151.184
C04334=1105.382,308.974,419.728,-179.994,15.168,151.185
C04335=1105.375,308.726,419.759,-179.998,15.166,151.185
C04336=1105.370,308.478,419.790,179.999,15.165,151.186
C04337=1105.364,308.231,419.820,179.995,15.164,151.186
C04338=1105.359,307.983,419.852,179.992,15.163,151.187
C04339=1105.352,307.734,419.883,179.988,15.161,151.187
C04340=1105.347,307.486,419.914,179.984,15.160,151.188
C04341=1105.342,307.239,419.945,179.981,15.159,151.188
C04342=1105.336,306.991,419.976,179.977,15.157,151.188
C04343=1105.329,306.742,420.006,179.973,15.155,151.189
C04344=1105.324,306.494,420.037,179.970,15.155,151.189
C04345=1105.318,306.247,420.068,179.966,15.153,151.190
C04346=1105.313,305.999,420.099,179.962,15.152,151.190
C04347=1105.307,305.751,420.130,179.959,15.150,151.191
C04348=1105.302,305.502,420.161,179.955,15.149,151.191
C04349=1105.296,305.255,420.191,179.951,15.147,151.192
C04350=1105.290,305.007,420.223,179.948,15.147,151.192
C04351=1105.285,304.759,420.253,179.944,15.145,151.193
C04352=1105.280,304.511,420.284,179.941,15.144,151.193
C04353=1105.273,304.263,420.315,179.938,15.142,151.194
C04354=1105.268,304.014,420.346,179.934,15.141,151.194
C04355=1105.262,303.767,420.376,179.930,15.140,151.195
C04356=1105.254,303.388,420.423,179.924,15.138,151.195
C04357=1105.245,303.008,420.471,179.919,15.136,151.196
C04358=1105.236,302.629,420.517,179.914,15.134,151.197
C04359=1105.228,302.250,420.564,179.908,15.133,151.198
C04360=1105.223,302.002,420.595,179.904,15.131,151.198
C04361=1105.217,301.754,420.625,179.901,15.130,151.199
C04362=1105.210,301.505,420.656,179.898,15.128,151.199
C04363=1105.205,301.257,420.687,179.894,15.127,151.199
C04364=1105.200,301.009,420.717,179.891,15.126,151.200
C04365=1105.194,300.762,420.748,179.887,15.125,151.200
C04366=1105.189,300.513,420.779,179.883,15.123,151.201
C04367=1105.183,300.266,420.809,179.879,15.122,151.201
C04368=1105.177,300.017,420.838,179.876,15.121,151.202
C04369=1105.172,299.769,420.869,179.872,15.120,151.202
C04370=1105.166,299.521,420.900,179.868,15.119,151.203
C04371=1105.161,299.273,420.930,179.865,15.118,151.203
C04372=1105.156,299.025,420.961,179.861,15.116,151.204
C04373=1105.150,298.777,420.991,179.857,15.115,151.204
C04374=1105.144,298.529,421.021,179.854,15.114,151.205
C04375=1105.138,298.281,421.051,179.850,15.113,151.205
C04376=1105.133,298.033,421.082,179.847,15.112,151.206
C04377=1105.128,297.785,421.113,179.843,15.110,151.206
C04378=1105.122,297.537,421.143,179.840,15.110,151.207
C04379=1105.116,297.289,421.173,179.836,15.108,151.208
C04380=1105.110,297.041,421.203,179.833,15.108,151.208
C04381=1105.105,296.793,421.233,179.829,15.106,151.209
C04382=1105.098,296.545,421.264,179.825,15.105,151.209
C04383=1105.093,296.296,421.294,179.821,15.104,151.210
C04384=1105.088,296.048,421.325,179.818,15.103,151.210
C04385=1105.082,295.800,421.355,179.814,15.102,151.211
C04386=1105.076,295.552,421.385,179.810,15.101,151.211
C04387=1105.070,295.304,421.415,179.807,15.100,151.212
C04388=1105.065,295.056,421.445,179.803,15.098,151.212
C04389=1105.059,294.808,421.475,179.800,15.098,151.213
C04390=1105.053,294.560,421.505,179.796,15.097,151.214
C04391=1105.048,294.312,421.535,179.792,15.096,151.214
C04392=1105.042,294.064,421.565,179.788,15.094,151.215
C04393=1105.036,293.815,421.595,179.785,15.093,151.215
C04394=1105.031,293.568,421.625,179.781,15.092,151.216
C04395=1105.025,293.319,421.655,179.778,15.092,151.216
C04396=1105.019,293.071,421.685,179.774,15.090,151.217
C04397=1105.014,292.823,421.715,179.771,15.089,151.217
C04398=1105.008,292.575,421.745,179.766,15.088,151.218
C04399=1105.003,292.327,421.775,179.763,15.088,151.218
C04400=1104.997,292.079,421.805,179.759,15.086,151.219
C04401=1104.992,291.831,421.835,179.756,15.086,151.220
C04402=1104.985,291.583,421.864,179.752,15.084,151.220
C04403=1104.980,291.335,421.894,179.749,15.083,151.221
C04404=1104.974,291.087,421.924,179.744,15.082,151.221
C04405=1104.968,290.839,421.954,179.741,15.082,151.222
C04406=1104.963,290.590,421.984,179.737,15.080,151.222
C04407=1104.957,290.343,422.014,179.734,15.080,151.223
C04408=1104.949,289.977,422.057,179.728,15.078,151.224
C04409=1104.941,289.612,422.102,179.722,15.076,151.225
C04410=1104.932,289.246,422.146,179.717,15.075,151.226
C04411=1104.923,288.880,422.189,179.712,15.074,151.226
C04412=1104.918,288.632,422.219,179.708,15.073,151.227
C04413=1104.911,288.384,422.248,179.704,15.072,151.228
C04414=1104.906,288.137,422.278,179.701,15.071,151.228
C04415=1104.901,287.888,422.307,179.697,15.070,151.229
C04416=1104.895,287.640,422.337,179.694,15.069,151.229
C04417=1104.889,287.392,422.367,179.689,15.068,151.230
C04418=1104.883,287.144,422.396,179.686,15.068,151.231
C04419=1104.878,286.895,422.426,179.683,15.067,151.231
C04420=1104.872,286.647,422.456,179.679,15.066,151.232
C04421=1104.866,286.399,422.485,179.675,15.065,151.232
C04422=1104.861,286.151,422.514,179.671,15.064,151.233
C04423=1104.856,285.903,422.543,179.668,15.063,151.234
C04424=1104.849,285.655,422.573,179.664,15.062,151.234
C04425=1104.844,285.407,422.603,179.660,15.062,151.235
C04426=1104.838,285.158,422.633,179.656,15.060,151.235
C04427=1104.833,284.910,422.662,179.653,15.060,151.236
C04428=1104.827,284.662,422.691,179.650,15.059,151.236
C04429=1104.821,284.414,422.720,179.645,15.058,151.237
C04430=1104.816,284.165,422.750,179.642,15.057,151.238
C04431=1104.810,283.917,422.779,179.638,15.056,151.238
C04432=1104.804,283.669,422.809,179.635,15.055,151.239
C04433=1104.799,283.421,422.837,179.630,15.054,151.240
C04434=1104.793,283.173,422.867,179.627,15.054,151.240
C04435=1104.787,282.925,422.897,179.624,15.053,151.241
C04436=1104.781,282.676,422.926,179.619,15.052,151.241
C04437=1104.776,282.429,422.955,179.616,15.051,151.242
C04438=1104.771,282.180,422.985,179.612,15.050,151.243
C04439=1104.765,281.932,423.014,179.609,15.050,151.243
C04440=1104.759,281.683,423.043,179.604,15.049,151.244
C04441=1104.754,281.436,423.071,179.601,15.048,151.244
C04442=1104.748,281.187,423.101,179.598,15.047,151.245
C04443=1104.742,280.939,423.130,179.594,15.046,151.246
C04444=1104.736,280.691,423.160,179.590,15.046,151.246
C04445=1104.731,280.443,423.188,179.586,15.045,151.247
C04446=1104.726,280.194,423.217,179.583,15.044,151.248
C04447=1104.719,279.946,423.246,179.579,15.043,151.248
C04448=1104.714,279.698,423.276,179.575,15.042,151.249
C04449=1104.708,279.450,423.305,179.572,15.042,151.249
C04450=1104.703,279.202,423.334,179.567,15.041,151.250
C04451=1104.697,278.953,423.362,179.564,15.040,151.251
C04452=1104.691,278.704,423.392,179.561,15.040,151.251
C04453=1104.686,278.457,423.421,179.556,15.039,151.252
C04454=1104.680,278.208,423.449,179.553,15.038,151.253
C04455=1104.674,277.960,423.479,179.549,15.037,151.253
C04456=1104.668,277.712,423.507,179.545,15.037,151.254
C04457=1104.663,277.463,423.536,179.542,15.036,151.255
C04458=1104.657,277.215,423.565,179.538,15.035,151.255
C04459=1104.651,276.968,423.594,179.534,15.035,151.256
C04460=1104.643,276.611,423.635,179.529,15.033,151.257
C04461=1104.635,276.255,423.677,179.523,15.032,151.258
C04462=1104.627,275.899,423.718,179.518,15.031,151.259
C04463=1104.619,275.543,423.759,179.513,15.031,151.260
C04464=1104.613,275.295,423.789,179.509,15.029,151.260
C04465=1104.608,275.047,423.817,179.506,15.029,151.261
C04466=1104.602,274.798,423.846,179.501,15.028,151.262
C04467=1104.596,274.550,423.875,179.498,15.028,151.262
C04468=1104.591,274.302,423.903,179.494,15.027,151.263
C04469=1104.585,274.054,423.932,179.490,15.026,151.263
C04470=1104.579,273.806,423.960,179.487,15.026,151.264
C04471=1104.574,273.557,423.989,179.483,15.025,151.265
C04472=1104.568,273.309,424.018,179.479,15.024,151.265
C04473=1104.563,273.060,424.046,179.476,15.024,151.266
C04474=1104.556,272.812,424.075,179.472,15.023,151.267
C04475=1104.551,272.563,424.104,179.468,15.022,151.268
C04476=1104.546,272.315,424.132,179.465,15.022,151.268
C04477=1104.540,272.067,424.161,179.461,15.021,151.269
C04478=1104.534,271.819,424.189,179.457,15.020,151.269
C04479=1104.528,271.571,424.218,179.453,15.020,151.270
C04480=1104.523,271.323,424.246,179.450,15.020,151.271
C04481=1104.517,271.074,424.275,179.445,15.019,151.271
C04482=1104.511,270.826,424.304,179.442,15.018,151.272
C04483=1104.506,270.578,424.332,179.438,15.017,151.273
C04484=1104.500,270.329,424.360,179.434,15.016,151.273
C04485=1104.494,270.081,424.388,179.431,15.016,151.274
C04486=1104.488,269.833,424.417,179.427,15.015,151.275
C04487=1104.483,269.585,424.445,179.423,15.015,151.275
C04488=1104.477,269.336,424.474,179.420,15.014,151.276
C04489=1104.472,269.088,424.502,179.416,15.014,151.277
C04490=1104.466,268.839,424.531,179.412,15.013,151.278
C04491=1104.460,268.591,424.560,179.408,15.013,151.278
C04492=1104.455,268.343,424.588,179.405,15.012,151.279
C04493=1104.449,268.094,424.616,179.400,15.011,151.280
C04494=1104.444,267.846,424.644,179.397,15.011,151.280
C04495=1104.438,267.597,424.672,179.393,15.011,151.281
C04496=1104.432,267.349,424.700,179.389,15.010,151.282
C04497=1104.426,267.100,424.728,179.386,15.009,151.282
C04498=1104.421,266.853,424.757,179.382,15.009,151.283
C04499=1104.415,266.604,424.785,179.378,15.008,151.284
C04500=1104.409,266.356,424.813,179.374,15.008,151.284
C04501=1104.403,266.107,424.842,179.371,15.007,151.285
C04502=1104.398,265.859,424.870,179.366,15.006,151.286
C04503=1104.392,265.610,424.898,179.363,15.006,151.287
C04504=1104.387,265.362,424.926,179.359,15.006,151.287
C04505=1104.381,265.114,424.954,179.356,15.005,151.288
C04506=1104.376,264.866,424.982,179.352,15.004,151.289
C04507=1104.370,264.618,425.010,179.348,15.004,151.289
C04508=1104.364,264.369,425.038,179.345,15.004,151.290
C04509=1104.358,264.121,425.066,179.340,15.003,151.291
C04510=1104.352,263.872,425.094,179.337,15.002,151.291
C04511=1104.347,263.624,425.122,179.333,15.002,151.292
C04512=1104.339,263.271,425.162,179.328,15.001,151.293
C04513=1104.330,262.917,425.201,179.323,15.001,151.294
C04514=1104.322,262.565,425.241,179.317,15.000,151.295
C04515=1104.314,262.211,425.281,179.311,14.999,151.296
C04516=1104.308,261.963,425.309,179.308,14.999,151.297
C04517=1104.302,261.714,425.336,179.304,14.999,151.298
C04518=1104.297,261.466,425.364,179.300,14.998,151.298
C04519=1104.291,261.218,425.392,179.296,14.998,151.299
C04520=1104.285,260.969,425.420,179.293,14.997,151.300
C04521=1104.279,260.721,425.447,179.289,14.997,151.301
C04522=1104.274,260.472,425.475,179.285,14.996,151.301
C04523=1104.268,260.224,425.503,179.281,14.996,151.302
C04524=1104.262,259.976,425.530,179.277,14.996,151.303
C04525=1104.256,259.727,425.559,179.274,14.995,151.304
C04526=1104.251,259.479,425.586,179.270,14.994,151.304
C04527=1104.245,259.230,425.614,179.266,14.994,151.305
C04528=1104.239,258.982,425.642,179.262,14.994,151.306
C04529=1104.234,258.734,425.669,179.259,14.994,151.306
C04530=1104.227,258.485,425.697,179.254,14.993,151.307
C04531=1104.222,258.237,425.725,179.251,14.993,151.308
C04532=1104.217,257.988,425.752,179.247,14.992,151.309
C04533=1104.210,257.740,425.780,179.244,14.992,151.309
C04534=1104.205,257.491,425.807,179.239,14.991,151.310
C04535=1104.200,257.243,425.835,179.236,14.991,151.311
C04536=1104.193,256.995,425.862,179.232,14.991,151.312
C04537=1104.188,256.746,425.890,179.229,14.990,151.312
C04538=1104.183,256.498,425.918,179.224,14.989,151.313
C04539=1104.177,256.249,425.945,179.220,14.989,151.314
C04540=1104.171,256.001,425.973,179.217,14.989,151.314
C04541=1104.165,255.753,425.999,179.213,14.989,151.315
C04542=1104.159,255.504,426.028,179.209,14.988,151.316
C04543=1104.154,255.256,426.054,179.206,14.987,151.317
C04544=1104.148,255.007,426.082,179.202,14.988,151.317
C04545=1104.143,254.759,426.109,179.198,14.987,151.318
C04546=1104.137,254.510,426.137,179.194,14.986,151.319
C04547=1104.132,254.262,426.164,179.190,14.986,151.320
C04548=1104.126,254.013,426.191,179.187,14.986,151.320
C04549=1104.120,253.765,426.219,179.183,14.986,151.321
C04550=1104.114,253.516,426.246,179.179,14.985,151.322
C04551=1104.109,253.268,426.274,179.175,14.984,151.322
C04552=1104.103,253.020,426.301,179.172,14.984,151.323
C04553=1104.098,252.771,426.328,179.168,14.984,151.324
C04554=1104.092,252.523,426.355,179.164,14.984,151.325
C04555=1104.086,252.274,426.383,179.160,14.983,151.325
C04556=1104.080,252.026,426.409,179.156,14.983,151.326
C04557=1104.075,251.777,426.437,179.153,14.982,151.327
C04558=1104.069,251.529,426.464,179.149,14.982,151.328
C04559=1104.064,251.281,426.491,179.145,14.982,151.328
C04560=1104.058,251.032,426.518,179.141,14.981,151.329
C04561=1104.053,250.783,426.546,179.138,14.981,151.330
C04562=1104.047,250.535,426.573,179.134,14.981,151.331
C04563=1104.042,250.286,426.600,179.130,14.981,151.331
C04564=1104.034,249.931,426.639,179.125,14.980,151.332
C04565=1104.025,249.575,426.678,179.120,14.980,151.333
C04566=1104.018,249.219,426.716,179.114,14.979,151.335
C04567=1104.009,248.862,426.755,179.108,14.978,151.336
C04568=1104.004,248.614,426.782,179.105,14.978,151.336
C04569=1103.998,248.366,426.810,179.101,14.978,151.337
C04570=1103.993,248.117,426.836,179.097,14.978,151.338
C04571=1103.988,247.869,426.864,179.094,14.977,151.339
C04572=1103.982,247.620,426.890,179.090,14.976,151.339
C04573=1103.976,247.372,426.917,179.086,14.976,151.340
C04574=1103.971,247.123,426.944,179.082,14.976,151.341
C04575=1103.965,246.875,426.971,179.079,14.976,151.342
C04576=1103.959,246.626,426.998,179.075,14.976,151.342
C04577=1103.953,246.377,427.024,179.070,14.975,151.343
C04578=1103.948,246.129,427.052,179.067,14.975,151.344
C04579=1103.942,245.880,427.078,179.063,14.975,151.345
C04580=1103.936,245.632,427.105,179.060,14.974,151.345
C04581=1103.931,245.384,427.132,179.056,14.974,151.346
C04582=1103.926,245.135,427.159,179.052,14.974,151.347
C04583=1103.920,244.887,427.186,179.048,14.973,151.348
C04584=1103.914,244.638,427.212,179.044,14.973,151.348
C04585=1103.908,244.390,427.239,179.040,14.973,151.349
C04586=1103.904,244.141,427.265,179.037,14.973,151.350
C04587=1103.898,243.892,427.292,179.033,14.973,151.351
C04588=1103.892,243.644,427.319,179.029,14.973,151.352
C04589=1103.886,243.396,427.345,179.025,14.972,151.352
C04590=1103.880,243.147,427.372,179.022,14.971,151.353
C04591=1103.874,242.898,427.399,179.018,14.972,151.354
C04592=1103.868,242.650,427.426,179.014,14.971,151.355
C04593=1103.864,242.400,427.452,179.010,14.971,151.355
C04594=1103.858,242.152,427.479,179.007,14.971,151.356
C04595=1103.852,241.904,427.505,179.003,14.970,151.357
C04596=1103.846,241.655,427.532,178.999,14.970,151.358
C04597=1103.841,241.406,427.558,178.995,14.970,151.358
C04598=1103.835,241.158,427.585,178.991,14.970,151.359
C04599=1103.829,240.910,427.611,178.988,14.970,151.360
C04600=1103.823,240.661,427.638,178.984,14.970,151.361
C04601=1103.818,240.412,427.664,178.980,14.970,151.362
C04602=1103.812,240.164,427.691,178.976,14.969,151.362
C04603=1103.806,239.916,427.717,178.972,14.969,151.363
C04604=1103.801,239.667,427.743,178.969,14.968,151.364
C04605=1103.795,239.418,427.770,178.965,14.969,151.365
C04606=1103.789,239.170,427.796,178.961,14.968,151.365
C04607=1103.784,238.921,427.822,178.957,14.968,151.366
C04608=1103.778,238.673,427.849,178.954,14.968,151.367
C04609=1103.772,238.424,427.876,178.950,14.968,151.368
C04610=1103.767,238.175,427.902,178.946,14.967,151.369
C04611=1103.761,237.927,427.928,178.942,14.967,151.369
C04612=1103.756,237.678,427.954,178.938,14.967,151.370
C04613=1103.750,237.430,427.981,178.935,14.967,151.371
C04614=1103.744,237.181,428.006,178.931,14.967,151.372
C04615=1103.738,236.933,428.033,178.927,14.967,151.372
C04616=1103.730,236.569,428.071,178.921,14.966,151.374
C04617=1103.722,236.207,428.110,178.916,14.966,151.375
C04618=1103.714,235.845,428.148,178.910,14.966,151.376
C04619=1103.706,235.482,428.186,178.905,14.966,151.377
C04620=1103.700,235.233,428.212,178.902,14.966,151.378
C04621=1103.694,234.984,428.238,178.897,14.965,151.379
C04622=1103.689,234.736,428.264,178.893,14.965,151.379
C04623=1103.684,234.488,428.290,178.890,14.965,151.380
C04624=1103.677,234.239,428.316,178.886,14.965,151.381
C04625=1103.672,233.991,428.342,178.882,14.965,151.382
C04626=1103.666,233.742,428.368,178.879,14.965,151.383
C04627=1103.661,233.493,428.394,178.875,14.965,151.383
C04628=1103.655,233.245,428.421,178.871,14.965,151.384
C04629=1103.649,232.996,428.446,178.868,14.965,151.385
C04630=1103.644,232.748,428.472,178.864,14.965,151.386
C04631=1103.638,232.499,428.499,178.860,14.964,151.387
C04632=1103.633,232.250,428.524,178.856,14.964,151.387
C04633=1103.626,232.002,428.550,178.852,14.964,151.388
C04634=1103.621,231.753,428.576,178.848,14.964,151.389
C04635=1103.615,231.504,428.602,178.845,14.963,151.390
C04636=1103.610,231.256,428.628,178.841,14.964,151.391
C04637=1103.604,231.007,428.653,178.837,14.963,151.391
C04638=1103.599,230.758,428.679,178.833,14.963,151.392
C04639=1103.593,230.510,428.706,178.830,14.963,151.393
C04640=1103.587,230.261,428.731,178.826,14.963,151.394
C04641=1103.581,230.012,428.757,178.822,14.963,151.394
C04642=1103.576,229.764,428.783,178.819,14.963,151.395
C04643=1103.570,229.515,428.808,178.814,14.962,151.396
C04644=1103.565,229.266,428.834,178.810,14.962,151.397
C04645=1103.558,229.018,428.860,178.807,14.963,151.398
C04646=1103.553,228.769,428.886,178.803,14.962,151.399
C04647=1103.548,228.521,428.912,178.799,14.962,151.399
C04648=1103.542,228.272,428.937,178.796,14.962,151.400
C04649=1103.536,228.023,428.963,178.792,14.962,151.401
C04650=1103.530,227.775,428.988,178.788,14.962,151.402
C04651=1103.524,227.526,429.014,178.784,14.962,151.403
C04652=1103.519,227.278,429.039,178.780,14.962,151.403
C04653=1103.513,227.029,429.065,178.777,14.962,151.404
C04654=1103.507,226.780,429.090,178.773,14.962,151.405
C04655=1103.502,226.531,429.116,178.769,14.962,151.406
C04656=1103.497,226.283,429.142,178.766,14.962,151.407
C04657=1103.491,226.034,429.167,178.762,14.962,151.407
C04658=1103.485,225.785,429.193,178.758,14.962,151.408
C04659=1103.480,225.537,429.218,178.754,14.962,151.409
C04660=1103.474,225.288,429.244,178.750,14.961,151.410
C04661=1103.468,225.040,429.269,178.746,14.961,151.411
C04662=1103.462,224.791,429.295,178.743,14.961,151.411
C04663=1103.457,224.543,429.320,178.739,14.961,151.412
C04664=1103.451,224.294,429.346,178.735,14.961,151.413
C04665=1103.445,224.045,429.371,178.731,14.961,151.414
C04666=1103.440,223.796,429.396,178.727,14.961,151.415
C04667=1103.434,223.547,429.422,178.724,14.961,151.416
C04668=1103.426,223.177,429.459,178.719,14.962,151.417
C04669=1103.418,222.806,429.498,178.713,14.961,151.418
C04670=1103.409,222.435,429.535,178.707,14.962,151.419
C04671=1103.401,222.063,429.573,178.702,14.961,151.420
C04672=1103.395,221.814,429.598,178.698,14.961,151.421
C04673=1103.390,221.566,429.624,178.694,14.961,151.422
C04674=1103.384,221.317,429.649,178.690,14.961,151.423
C04675=1103.378,221.068,429.674,178.686,14.961,151.424
C04676=1103.372,220.820,429.699,178.683,14.961,151.425
C04677=1103.367,220.571,429.725,178.679,14.961,151.425
C04678=1103.361,220.322,429.749,178.675,14.961,151.426
C04679=1103.355,220.074,429.774,178.672,14.961,151.427
C04680=1103.350,219.825,429.800,178.668,14.961,151.428
C04681=1103.344,219.576,429.826,178.664,14.961,151.429
C04682=1103.338,219.328,429.850,178.660,14.961,151.429
C04683=1103.332,219.079,429.875,178.656,14.961,151.430
C04684=1103.328,218.830,429.900,178.653,14.961,151.431
C04685=1103.321,218.581,429.925,178.649,14.961,151.432
C04686=1103.315,218.333,429.951,178.645,14.961,151.433
C04687=1103.310,218.084,429.975,178.641,14.962,151.434
C04688=1103.304,217.835,430.000,178.638,14.961,151.434
C04689=1103.299,217.587,430.025,178.634,14.961,151.435
C04690=1103.293,217.338,430.050,178.630,14.961,151.436
C04691=1103.287,217.090,430.075,178.626,14.961,151.437
C04692=1103.281,216.841,430.100,178.623,14.962,151.438
C04693=1103.276,216.593,430.125,178.619,14.961,151.438
C04694=1103.271,216.343,430.150,178.615,14.962,151.439
C04695=1103.264,216.094,430.176,178.611,14.962,151.440
C04696=1103.259,215.846,430.200,178.608,14.961,151.441
C04697=1103.253,215.597,430.225,178.604,14.962,151.442
C04698=1103.248,215.349,430.249,178.600,14.961,151.443
C04699=1103.242,215.099,430.275,178.596,14.962,151.443
C04700=1103.237,214.851,430.300,178.593,14.962,151.444
C04701=1103.231,214.602,430.324,178.589,14.962,151.445
C04702=1103.225,214.354,430.349,178.585,14.962,151.446
C04703=1103.219,214.104,430.374,178.582,14.961,151.447
C04704=1103.214,213.856,430.398,178.578,14.962,151.447
C04705=1103.209,213.608,430.423,178.574,14.962,151.448
C04706=1103.203,213.359,430.448,178.570,14.962,151.449
C04707=1103.197,213.111,430.473,178.566,14.962,151.450
C04708=1103.191,212.861,430.497,178.563,14.962,151.451
C04709=1103.187,212.612,430.522,178.559,14.962,151.452
C04710=1103.180,212.364,430.547,178.555,14.962,151.452
C04711=1103.175,212.115,430.572,178.551,14.962,151.453
C04712=1103.169,211.866,430.596,178.548,14.962,151.454
C04713=1103.164,211.617,430.621,178.544,14.962,151.455
C04714=1103.158,211.369,430.646,178.540,14.962,151.456
C04715=1103.152,211.120,430.670,178.536,14.962,151.457
C04716=1103.146,210.871,430.695,178.533,14.962,151.457
C04717=1103.140,210.623,430.718,178.529,14.962,151.458
C04718=1103.135,210.375,430.743,178.525,14.962,151.459
C04719=1103.129,210.125,430.768,178.521,14.962,151.460
C04720=1103.121,209.758,430.805,178.516,14.963,151.461
C04721=1103.112,209.390,430.841,178.511,14.963,151.462
C04722=1103.104,209.022,430.877,178.505,14.963,151.464
C04723=1103.096,208.655,430.913,178.499,14.963,151.465
C04724=1103.073,207.654,431.010,178.468,14.958,151.471
C04725=1103.067,207.405,431.035,178.464,14.959,151.472
C04726=1103.062,207.156,431.059,178.460,14.960,151.473
C04727=1103.056,206.908,431.083,178.456,14.961,151.474
C04728=1103.050,206.659,431.107,178.452,14.962,151.475
C04729=1103.045,206.410,431.132,178.448,14.963,151.476
C04730=1103.039,206.162,431.156,178.444,14.964,151.477
C04731=1103.033,205.913,431.180,178.440,14.965,151.478
C04732=1103.027,205.664,431.204,178.436,14.965,151.479
C04733=1103.022,205.416,431.229,178.432,14.967,151.480
C04734=1103.016,205.166,431.253,178.428,14.967,151.481
C04735=1103.010,204.918,431.277,178.424,14.968,151.482
C04736=1103.005,204.669,431.301,178.421,14.969,151.483
C04737=1102.999,204.420,431.326,178.416,14.970,151.484
C04738=1102.993,204.171,431.349,178.412,14.971,151.486
C04739=1102.988,203.923,431.373,178.408,14.972,151.487
C04740=1102.983,203.674,431.397,178.404,14.973,151.488
C04741=1102.976,203.425,431.421,178.400,14.973,151.489
C04742=1102.971,203.176,431.445,178.396,14.975,151.490
C04743=1102.965,202.928,431.470,178.392,14.975,151.491
C04744=1102.959,202.678,431.493,178.388,14.976,151.492
C04745=1102.954,202.430,431.517,178.385,14.977,151.493
C04746=1102.948,202.181,431.541,178.380,14.978,151.494
C04747=1102.942,201.933,431.565,178.376,14.979,151.495
C04748=1102.936,201.684,431.589,178.373,14.980,151.496
C04749=1102.931,201.435,431.613,178.369,14.981,151.497
C04750=1102.925,201.186,431.636,178.364,14.981,151.498
C04751=1102.919,200.937,431.661,178.361,14.983,151.499
C04752=1102.913,200.688,431.684,178.357,14.983,151.500
C04753=1102.908,200.440,431.708,178.353,14.985,151.502
C04754=1102.902,200.191,431.732,178.349,14.986,151.503
C04755=1102.896,199.942,431.757,178.345,14.986,151.504
C04756=1102.890,199.693,431.779,178.341,14.988,151.505
C04757=1102.885,199.445,431.804,178.337,14.988,151.506
C04758=1102.879,199.196,431.827,178.333,14.989,151.507
C04759=1102.873,198.946,431.851,178.329,14.990,151.508
C04760=1102.867,198.698,431.875,178.325,14.991,151.509
C04761=1102.862,198.449,431.898,178.321,14.991,151.510
C04762=1102.856,198.201,431.922,178.317,14.993,151.511
C04763=1102.850,197.952,431.946,178.313,14.993,151.512
C04764=1102.845,197.702,431.970,178.309,14.994,151.513
C04765=1102.838,197.454,431.993,178.306,14.995,151.514
C04766=1102.833,197.205,432.017,178.302,14.996,151.515
C04767=1102.827,196.957,432.041,178.298,14.996,151.516
C04768=1102.822,196.708,432.064,178.294,14.998,151.517
C04769=1102.816,196.458,432.088,178.290,14.998,151.518
C04770=1102.810,196.210,432.111,178.286,14.999,151.519
C04771=1102.805,195.961,432.135,178.282,15.000,151.520
C04772=1102.799,195.712,432.158,178.278,15.001,151.521
C04773=1102.793,195.464,432.182,178.274,15.002,151.523
C04774=1102.788,195.215,432.205,178.270,15.003,151.524
C04775=1102.781,194.966,432.230,178.266,15.003,151.524
C04776=1102.776,194.717,432.252,178.263,15.004,151.526
C04777=1102.770,194.468,432.277,178.259,15.005,151.527
C04778=1102.765,194.219,432.300,178.255,15.006,151.528
C04779=1102.759,193.970,432.323,178.251,15.007,151.529
C04780=1102.754,193.722,432.347,178.247,15.008,151.530
C04781=1102.748,193.473,432.370,178.243,15.008,151.531
C04782=1102.742,193.225,432.393,178.240,15.009,151.532
C04783=1102.737,192.975,432.417,178.235,15.010,151.533
C04784=1102.731,192.726,432.440,178.231,15.011,151.534
C04785=1102.725,192.454,432.466,178.227,15.011,151.535
C04786=1102.718,192.182,432.491,178.223,15.013,151.536
C04787=1102.712,191.910,432.518,178.219,15.014,151.537
C04788=1102.706,191.638,432.542,178.215,15.015,151.538
C04789=1102.700,191.389,432.565,178.211,15.015,151.539
C04790=1102.695,191.141,432.589,178.206,15.016,151.540
C04791=1102.689,190.892,432.612,178.203,15.017,151.541
C04792=1102.684,190.643,432.635,178.199,15.017,151.542
C04793=1102.679,190.394,432.659,178.196,15.019,151.543
C04794=1102.673,190.145,432.683,178.192,15.019,151.544
C04795=1102.667,189.897,432.705,178.188,15.020,151.545
C04796=1102.661,189.648,432.728,178.184,15.021,151.546
C04797=1102.656,189.398,432.752,178.180,15.021,151.547
C04798=1102.650,189.150,432.775,178.176,15.022,151.548
C04799=1102.645,188.901,432.798,178.173,15.023,151.549
C04800=1102.639,188.652,432.822,178.169,15.024,151.550
C04801=1102.633,188.403,432.844,178.165,15.024,151.551
C04802=1102.628,188.154,432.868,178.161,15.026,151.552
C04803=1102.622,187.905,432.891,178.157,15.026,151.553
C04804=1102.617,187.656,432.914,178.153,15.027,151.554
C04805=1102.611,187.408,432.937,178.150,15.028,151.555
C04806=1102.605,187.159,432.960,178.146,15.028,151.556
C04807=1102.600,186.909,432.983,178.142,15.029,151.557
C04808=1102.594,186.661,433.006,178.138,15.030,151.558
C04809=1102.589,186.412,433.029,178.134,15.030,151.559
C04810=1102.583,186.163,433.052,178.131,15.031,151.560
C04811=1102.577,185.914,433.075,178.127,15.032,151.561
C04812=1102.571,185.665,433.098,178.123,15.032,151.562
C04813=1102.567,185.416,433.121,178.120,15.034,151.563
C04814=1102.561,185.168,433.144,178.115,15.034,151.564
C04815=1102.556,184.919,433.167,178.111,15.035,151.565
C04816=1102.550,184.670,433.190,178.108,15.036,151.566
C04817=1102.543,184.421,433.212,178.104,15.037,151.567
C04818=1102.538,184.172,433.235,178.101,15.038,151.568
C04819=1102.532,183.923,433.258,178.096,15.038,151.569
C04820=1102.526,183.675,433.281,178.092,15.039,151.570
C04821=1102.520,183.426,433.304,178.089,15.040,151.571
C04822=1102.515,183.177,433.327,178.085,15.041,151.572
C04823=1102.509,182.928,433.350,178.081,15.041,151.573
C04824=1102.503,182.679,433.373,178.078,15.042,151.574
C04825=1102.497,182.430,433.395,178.073,15.043,151.575
C04826=1102.491,182.181,433.418,178.070,15.044,151.576
C04827=1102.485,181.933,433.441,178.066,15.044,151.577
C04828=1102.480,181.683,433.464,178.062,15.045,151.578
C04829=1102.474,181.434,433.486,178.059,15.046,151.579
C04830=1102.468,181.185,433.509,178.055,15.047,151.580
C04831=1102.462,180.937,433.532,178.051,15.048,151.581
C04832=1102.456,180.688,433.555,178.047,15.048,151.582
C04833=1102.451,180.438,433.577,178.043,15.049,151.583
C04834=1102.445,180.189,433.600,178.040,15.050,151.584
C04835=1102.439,179.940,433.623,178.036,15.051,151.585
C04836=1102.433,179.693,433.645,178.032,15.051,151.586
C04837=1102.428,179.444,433.668,178.028,15.052,151.587
C04838=1102.422,179.194,433.690,178.024,15.053,151.588
C04839=1102.417,178.945,433.713,178.021,15.054,151.589
C04840=1102.411,178.696,433.736,178.017,15.054,151.590
C04841=1102.405,178.447,433.758,178.013,15.055,151.591
C04842=1102.399,178.198,433.780,178.010,15.056,151.592
C04843=1102.393,177.949,433.803,178.006,15.057,151.593
C04844=1102.388,177.701,433.825,178.002,15.058,151.594
C04845=1102.382,177.452,433.848,177.998,15.058,151.595
C04846=1102.376,177.203,433.871,177.994,15.059,151.596
C04847=1102.371,176.954,433.893,177.991,15.059,151.597
C04848=1102.365,176.705,433.916,177.987,15.060,151.598
C04849=1102.359,176.433,433.940,177.983,15.061,151.599
C04850=1102.353,176.160,433.965,177.979,15.062,151.600
C04851=1102.346,175.888,433.990,177.976,15.063,151.601
C04852=1102.340,175.615,434.014,177.971,15.063,151.602
C04853=1102.334,175.367,434.036,177.967,15.064,151.603
C04854=1102.329,175.117,434.058,177.963,15.064,151.604
C04855=1102.323,174.869,434.081,177.960,15.065,151.605
C04856=1102.317,174.620,434.102,177.956,15.066,151.606
C04857=1102.312,174.371,434.125,177.953,15.067,151.607
C04858=1102.306,174.121,434.148,177.949,15.067,151.608
C04859=1102.300,173.873,434.170,177.945,15.068,151.609
C04860=1102.295,173.624,434.192,177.942,15.069,151.609
C04861=1102.289,173.375,434.215,177.938,15.069,151.610
C04862=1102.283,173.126,434.236,177.934,15.070,151.611
C04863=1102.278,172.878,434.259,177.930,15.071,151.612
C04864=1102.272,172.628,434.281,177.926,15.071,151.613
C04865=1102.266,172.379,434.303,177.923,15.072,151.614
C04866=1102.260,172.130,434.326,177.919,15.073,151.615
C04867=1102.256,171.881,434.348,177.916,15.074,151.616
C04868=1102.249,171.633,434.370,177.912,15.074,151.617
C04869=1102.244,171.383,434.392,177.908,15.074,151.618
C04870=1102.238,171.135,434.413,177.905,15.076,151.619
C04871=1102.232,170.886,434.436,177.901,15.076,151.620
C04872=1102.227,170.636,434.459,177.898,15.077,151.621
C04873=1102.221,170.388,434.480,177.894,15.077,151.622
C04874=1102.216,170.139,434.503,177.890,15.077,151.622
C04875=1102.210,169.890,434.525,177.887,15.078,151.623
C04876=1102.205,169.641,434.546,177.883,15.079,151.624
C04877=1102.199,169.392,434.569,177.879,15.079,151.625
C04878=1102.193,169.143,434.591,177.876,15.080,151.626
C04879=1102.188,168.894,434.613,177.872,15.081,151.627
C04880=1102.182,168.645,434.634,177.869,15.082,151.628
C04881=1102.176,168.396,434.657,177.865,15.082,151.629
C04882=1102.171,168.147,434.679,177.861,15.082,151.630
C04883=1102.165,167.898,434.701,177.858,15.083,151.631
C04884=1102.160,167.649,434.722,177.854,15.083,151.632
C04885=1102.154,167.400,434.744,177.851,15.084,151.633
C04886=1102.148,167.151,434.767,177.847,15.085,151.634
C04887=1102.143,166.902,434.789,177.843,15.085,151.634
C04888=1102.137,166.653,434.811,177.839,15.086,151.635
C04889=1102.132,166.404,434.832,177.836,15.087,151.636
C04890=1102.126,166.155,434.854,177.832,15.088,151.637
C04891=1102.121,165.906,434.876,177.829,15.088,151.638
C04892=1102.115,165.657,434.898,177.825,15.088,151.639
C04893=1102.109,165.408,434.920,177.822,15.089,151.640
C04894=1102.104,165.159,434.942,177.818,15.089,151.641
C04895=1102.098,164.910,434.964,177.815,15.090,151.642
C04896=1102.093,164.661,434.986,177.811,15.091,151.643
C04897=1102.087,164.412,435.007,177.807,15.091,151.643
C04898=1102.082,164.163,435.029,177.804,15.091,151.644
C04899=1102.076,163.914,435.051,177.800,15.092,151.645
C04900=1102.070,163.666,435.072,177.797,15.093,151.646
C04901=1102.065,163.416,435.094,177.793,15.093,151.647
C04902=1102.060,163.168,435.115,177.789,15.093,151.648
C04903=1102.054,162.918,435.138,177.786,15.094,151.649
C04904=1102.049,162.670,435.159,177.782,15.095,151.650
C04905=1102.043,162.420,435.181,177.779,15.096,151.650
C04906=1102.038,162.172,435.202,177.775,15.096,151.651
C04907=1102.032,161.922,435.225,177.772,15.096,151.652
C04908=1102.027,161.674,435.246,177.768,15.097,151.653
C04909=1102.020,161.424,435.268,177.765,15.097,151.654
C04910=1102.015,161.176,435.289,177.761,15.098,151.655
C04911=1102.009,160.926,435.311,177.758,15.098,151.656
C04912=1102.004,160.677,435.332,177.754,15.099,151.657
C04913=1101.997,160.404,435.355,177.750,15.100,151.658
C04914=1101.991,160.132,435.379,177.746,15.100,151.659
C04915=1101.985,159.859,435.403,177.742,15.101,151.659
C04916=1101.979,159.587,435.426,177.738,15.101,151.661
C04917=1101.973,159.337,435.448,177.734,15.102,151.661
C04918=1101.967,159.089,435.469,177.732,15.102,151.662
C04919=1101.962,158.839,435.491,177.728,15.103,151.663
C04920=1101.957,158.590,435.512,177.725,15.104,151.664
C04921=1101.950,158.341,435.533,177.721,15.104,151.665
C04922=1101.945,158.092,435.555,177.718,15.105,151.666
C04923=1101.939,157.843,435.576,177.714,15.105,151.667
C04924=1101.934,157.594,435.598,177.710,15.105,151.668
C04925=1101.928,157.345,435.619,177.707,15.106,151.668
C04926=1101.922,157.096,435.640,177.703,15.106,151.669
C04927=1101.916,156.847,435.662,177.700,15.107,151.670
C04928=1101.911,156.598,435.683,177.696,15.108,151.671
C04929=1101.905,156.349,435.704,177.693,15.109,151.672
C04930=1101.899,156.100,435.726,177.689,15.108,151.673
C04931=1101.894,155.851,435.747,177.685,15.109,151.674
C04932=1101.889,155.601,435.768,177.682,15.110,151.674
C04933=1101.883,155.353,435.790,177.678,15.110,151.675
C04934=1101.877,155.104,435.811,177.676,15.111,151.676
C04935=1101.872,154.855,435.832,177.672,15.111,151.677
C04936=1101.865,154.605,435.853,177.668,15.111,151.678
C04937=1101.860,154.357,435.875,177.665,15.112,151.679
C04938=1101.855,154.108,435.895,177.661,15.113,151.680
C04939=1101.849,153.859,435.917,177.658,15.113,151.680
C04940=1101.843,153.609,435.937,177.654,15.113,151.681
C04941=1101.837,153.360,435.959,177.651,15.114,151.682
C04942=1101.832,153.112,435.980,177.647,15.114,151.683
C04943=1101.826,152.863,436.001,177.644,15.115,151.684
C04944=1101.820,152.613,436.023,177.640,15.116,151.685
C04945=1101.815,152.364,436.043,177.637,15.115,151.685
C04946=1101.809,152.116,436.064,177.634,15.116,151.686
C04947=1101.803,151.866,436.085,177.630,15.117,151.687
C04948=1101.798,151.617,436.107,177.627,15.117,151.688
C04949=1101.792,151.368,436.127,177.623,15.118,151.689
C04950=1101.786,151.119,436.149,177.619,15.118,151.690
C04951=1101.781,150.870,436.169,177.616,15.118,151.691
C04952=1101.775,150.621,436.191,177.613,15.119,151.691
C04953=1101.770,150.372,436.211,177.610,15.119,151.692
C04954=1101.764,150.123,436.233,177.606,15.120,151.693
C04955=1101.758,149.873,436.254,177.603,15.121,151.694
C04956=1101.753,149.625,436.275,177.599,15.121,151.695
C04957=1101.748,149.376,436.295,177.595,15.121,151.696
C04958=1101.741,149.126,436.316,177.592,15.121,151.696
C04959=1101.735,148.878,436.337,177.589,15.122,151.697
C04960=1101.730,148.629,436.358,177.585,15.123,151.698
C04961=1101.725,148.380,436.379,177.582,15.123,151.699
C04962=1101.719,148.130,436.400,177.579,15.124,151.700
C04963=1101.713,147.881,436.420,177.575,15.123,151.701
C04964=1101.708,147.633,436.442,177.571,15.124,151.701
C04965=1101.701,147.383,436.462,177.568,15.124,151.702
C04966=1101.696,147.134,436.483,177.565,15.125,151.703
C04967=1101.690,146.885,436.504,177.562,15.125,151.704
C04968=1101.685,146.636,436.525,177.558,15.126,151.705
C04969=1101.679,146.387,436.545,177.555,15.126,151.705
C04970=1101.673,146.138,436.566,177.551,15.126,151.706
C04971=1101.667,145.888,436.587,177.548,15.127,151.707
C04972=1101.662,145.639,436.607,177.544,15.127,151.708
C04973=1101.657,145.390,436.628,177.541,15.127,151.709
C04974=1101.650,145.142,436.649,177.538,15.128,151.710
C04975=1101.645,144.892,436.670,177.534,15.128,151.710
C04976=1101.639,144.643,436.690,177.531,15.129,151.711
C04977=1101.633,144.370,436.713,177.527,15.129,151.712
C04978=1101.626,144.097,436.736,177.523,15.130,151.713
C04979=1101.621,143.824,436.758,177.520,15.130,151.714
C04980=1101.614,143.551,436.780,177.517,15.131,151.715
C04981=1101.609,143.302,436.801,177.513,15.131,151.716
C04982=1101.603,143.052,436.822,177.509,15.131,151.716
C04983=1101.597,142.804,436.842,177.506,15.131,151.717
C04984=1101.592,142.555,436.863,177.502,15.132,151.718
C04985=1101.587,142.306,436.883,177.500,15.132,151.719
C04986=1101.581,142.057,436.903,177.496,15.133,151.720
C04987=1101.575,141.807,436.924,177.493,15.133,151.720
C04988=1101.569,141.558,436.945,177.489,15.133,151.721
C04989=1101.563,141.309,436.965,177.487,15.134,151.722
C04990=1101.558,141.060,436.985,177.483,15.134,151.723
C04991=1101.553,140.811,437.006,177.479,15.134,151.723
C04992=1101.547,140.562,437.026,177.476,15.135,151.724
C04993=1101.541,140.312,437.047,177.472,15.135,151.725
C04994=1101.536,140.063,437.067,177.470,15.135,151.726
C04995=1101.530,139.814,437.087,177.466,15.135,151.727
C04996=1101.524,139.566,437.109,177.463,15.136,151.727
C04997=1101.518,139.317,437.129,177.459,15.136,151.728
C04998=1101.512,139.067,437.150,177.456,15.137,151.729
C04999=1101.507,138.818,437.169,177.453,15.137,151.730
C05000=1101.502,138.569,437.189,177.449,15.137,151.731
C05001=1101.496,138.320,437.210,177.446,15.138,151.731
C05002=1101.490,138.071,437.230,177.443,15.138,151.732
C05003=1101.485,137.822,437.250,177.439,15.139,151.733
C05004=1101.479,137.573,437.270,177.436,15.138,151.734
C05005=1101.473,137.323,437.291,177.433,15.139,151.734
C05006=1101.467,137.074,437.311,177.430,15.139,151.735
C05007=1101.462,136.825,437.332,177.426,15.140,151.736
C05008=1101.456,136.576,437.352,177.423,15.140,151.737
C05009=1101.451,136.327,437.372,177.420,15.140,151.738
C05010=1101.445,136.078,437.392,177.416,15.140,151.738
C05011=1101.440,135.829,437.412,177.413,15.140,151.739
C05012=1101.434,135.580,437.432,177.410,15.141,151.740
C05013=1101.428,135.331,437.452,177.406,15.141,151.741
C05014=1101.422,135.081,437.473,177.403,15.142,151.741
C05015=1101.416,134.832,437.493,177.400,15.142,151.742
C05016=1101.411,134.583,437.513,177.397,15.142,151.743
C05017=1101.405,134.334,437.533,177.393,15.142,151.744
C05018=1101.400,134.085,437.553,177.391,15.143,151.744
C05019=1101.394,133.836,437.573,177.387,15.143,151.745
C05020=1101.388,133.587,437.594,177.384,15.144,151.746
C05021=1101.382,133.338,437.614,177.380,15.143,151.747
C05022=1101.377,133.089,437.633,177.377,15.144,151.748
C05023=1101.371,132.839,437.654,177.374,15.144,151.748
C05024=1101.365,132.591,437.673,177.370,15.144,151.749
C05025=1101.361,132.341,437.693,177.368,15.144,151.750
C05026=1101.355,132.092,437.713,177.364,15.144,151.750
C05027=1101.349,131.843,437.733,177.361,15.145,151.751
C05028=1101.343,131.594,437.754,177.358,15.145,151.752
C05029=1101.338,131.345,437.773,177.355,15.145,151.753
C05030=1101.332,131.096,437.793,177.351,15.145,151.753
C05031=1101.325,130.846,437.813,177.348,15.146,151.754
C05032=1101.320,130.597,437.833,177.344,15.146,151.755
C05033=1101.314,130.348,437.853,177.342,15.147,151.756
C05034=1101.308,130.098,437.872,177.338,15.147,151.757
C05035=1101.302,129.850,437.892,177.335,15.147,151.757
C05036=1101.296,129.601,437.912,177.332,15.147,151.758
C05037=1101.291,129.351,437.932,177.329,15.148,151.759
C05038=1101.285,129.102,437.952,177.325,15.148,151.760
C05039=1101.279,128.853,437.972,177.322,15.148,151.760
C05040=1101.274,128.604,437.991,177.319,15.148,151.761
C05041=1101.268,128.331,438.013,177.315,15.148,151.762
C05042=1101.261,128.058,438.034,177.311,15.148,151.763
C05043=1101.256,127.784,438.056,177.309,15.149,151.763
C05044=1101.249,127.512,438.078,177.305,15.149,151.764
C05045=1101.243,127.263,438.098,177.301,15.149,151.765
C05046=1101.238,127.013,438.117,177.299,15.149,151.766
C05047=1101.232,126.764,438.137,177.295,15.149,151.766
C05048=1101.226,126.515,438.157,177.292,15.150,151.767
C05049=1101.220,126.266,438.177,177.289,15.150,151.768
C05050=1101.215,126.017,438.196,177.286,15.150,151.769
C05051=1101.209,125.767,438.215,177.282,15.150,151.769
C05052=1101.203,125.518,438.235,177.279,15.151,151.770
C05053=1101.198,125.269,438.255,177.276,15.151,151.771
C05054=1101.192,125.020,438.275,177.273,15.151,151.771
C05055=1101.186,124.770,438.294,177.270,15.151,151.772
C05056=1101.180,124.521,438.314,177.267,15.151,151.773
C05057=1101.175,124.272,438.333,177.263,15.151,151.774
C05058=1101.169,124.023,438.353,177.261,15.152,151.774
C05059=1101.163,123.774,438.373,177.257,15.152,151.775
C05060=1101.158,123.525,438.391,177.255,15.152,151.776
C05061=1101.153,123.275,438.411,177.251,15.152,151.776
C05062=1101.147,123.026,438.431,177.248,15.153,151.777
C05063=1101.141,122.777,438.450,177.245,15.152,151.778
C05064=1101.136,122.528,438.470,177.241,15.152,151.779
C05065=1101.130,122.279,438.490,177.238,15.153,151.779
C05066=1101.124,122.029,438.509,177.235,15.152,151.780
C05067=1101.118,121.780,438.528,177.232,15.153,151.781
C05068=1101.113,121.532,438.548,177.229,15.153,151.781
C05069=1101.107,121.282,438.567,177.226,15.153,151.782
C05070=1101.101,121.033,438.586,177.222,15.153,151.783
C05071=1101.096,120.784,438.605,177.220,15.154,151.784
C05072=1101.090,120.535,438.625,177.216,15.153,151.784
C05073=1101.084,120.285,438.645,177.214,15.154,151.785
C05074=1101.079,120.037,438.664,177.210,15.154,151.786
C05075=1101.073,119.787,438.683,177.207,15.154,151.786
C05076=1101.068,119.538,438.702,177.204,15.154,151.787
C05077=1101.062,119.289,438.722,177.201,15.154,151.788
C05078=1101.056,119.039,438.741,177.198,15.154,151.788
C05079=1101.051,118.791,438.760,177.195,15.154,151.789
C05080=1101.045,118.541,438.779,177.191,15.154,151.790
C05081=1101.040,118.292,438.799,177.189,15.154,151.790
C05082=1101.034,118.042,438.818,177.185,15.154,151.791
C05083=1101.028,117.793,438.837,177.183,15.154,151.792
C05084=1101.023,117.545,438.857,177.179,15.154,151.792
C05085=1101.017,117.295,438.876,177.176,15.155,151.793
C05086=1101.011,117.046,438.895,177.173,15.154,151.794
C05087=1101.006,116.797,438.914,177.170,15.155,151.794
C05088=1101.001,116.548,438.933,177.167,15.154,151.795
C05089=1100.995,116.298,438.953,177.164,15.155,151.796
C05090=1100.989,116.049,438.972,177.161,15.155,151.796
C05091=1100.984,115.800,438.991,177.158,15.155,151.797
C05092=1100.978,115.551,439.010,177.155,15.155,151.798
C05093=1100.973,115.301,439.029,177.152,15.155,151.798
C05094=1100.967,115.052,439.048,177.149,15.155,151.799
C05095=1100.962,114.803,439.067,177.145,15.155,151.800
C05096=1100.956,114.554,439.086,177.143,15.155,151.800
C05097=1100.951,114.304,439.106,177.139,15.155,151.801
C05098=1100.945,114.055,439.125,177.137,15.155,151.802
C05099=1100.939,113.807,439.143,177.133,15.155,151.802
C05100=1100.933,113.557,439.162,177.131,15.155,151.803
C05101=1100.928,113.308,439.182,177.127,15.155,151.804
C05102=1100.922,113.058,439.201,177.125,15.155,151.804
C05103=1100.917,112.809,439.220,177.121,15.155,151.805
C05104=1100.911,112.560,439.239,177.119,15.155,151.806
C05105=1100.904,112.287,439.259,177.115,15.155,151.806
C05106=1100.898,112.013,439.280,177.112,15.156,151.807
C05107=1100.892,111.741,439.301,177.109,15.156,151.808
C05108=1100.886,111.467,439.321,177.105,15.155,151.808
C05109=1100.880,111.218,439.340,177.102,15.156,151.809
C05110=1100.874,110.969,439.360,177.099,15.155,151.810
C05111=1100.869,110.720,439.378,177.096,15.156,151.810
C05112=1100.863,110.470,439.397,177.093,15.155,151.811
C05113=1100.858,110.221,439.416,177.090,15.156,151.812
C05114=1100.852,109.972,439.434,177.087,15.155,151.812
C05115=1100.846,109.723,439.453,177.084,15.156,151.813
C05116=1100.840,109.473,439.473,177.081,15.155,151.814
C05117=1100.834,109.224,439.490,177.078,15.156,151.814
C05118=1100.829,108.975,439.509,177.075,15.156,151.815
C05119=1100.823,108.725,439.529,177.072,15.156,151.816
C05120=1100.817,108.476,439.547,177.069,15.156,151.816
C05121=1100.812,108.228,439.566,177.066,15.156,151.817
C05122=1100.807,107.978,439.585,177.063,15.155,151.818
C05123=1100.800,107.728,439.603,177.060,15.156,151.818
C05124=1100.795,107.480,439.622,177.057,15.155,151.819
C05125=1100.789,107.230,439.640,177.054,15.155,151.819
C05126=1100.784,106.981,439.659,177.051,15.155,151.820
C05127=1100.778,106.732,439.678,177.048,15.156,151.821
C05128=1100.772,106.483,439.697,177.045,15.155,151.821
C05129=1100.767,106.233,439.715,177.042,15.156,151.822
C05130=1100.761,105.984,439.734,177.039,15.155,151.823
C05131=1100.755,105.735,439.753,177.037,15.155,151.823
C05132=1100.750,105.485,439.771,177.033,15.155,151.824
C05133=1100.744,105.236,439.790,177.030,15.155,151.825
C05134=1100.739,104.987,439.808,177.027,15.155,151.825
C05135=1100.732,104.738,439.827,177.025,15.155,151.826
C05136=1100.727,104.488,439.846,177.021,15.155,151.826
C05137=1100.721,104.239,439.863,177.019,15.155,151.827
C05138=1100.716,103.990,439.883,177.015,15.155,151.828
C05139=1100.711,103.741,439.901,177.013,15.155,151.828
C05140=1100.704,103.491,439.919,177.010,15.154,151.829
C05141=1100.699,103.243,439.938,177.007,15.154,151.829
C05142=1100.693,102.993,439.956,177.004,15.154,151.830
C05143=1100.688,102.744,439.975,177.001,15.154,151.831
C05144=1100.682,102.495,439.993,176.998,15.154,151.831
C05145=1100.676,102.245,440.012,176.995,15.154,151.832
C05146=1100.671,101.996,440.030,176.993,15.154,151.832
C05147=1100.665,101.747,440.049,176.989,15.154,151.833
C05148=1100.659,101.498,440.067,176.987,15.154,151.834
C05149=1100.654,101.248,440.086,176.984,15.153,151.834
C05150=1100.648,100.999,440.103,176.981,15.154,151.835
C05151=1100.643,100.750,440.123,176.978,15.154,151.836
C05152=1100.637,100.501,440.140,176.975,15.154,151.836
C05153=1100.631,100.251,440.158,176.972,15.153,151.837
C05154=1100.626,100.002,440.177,176.969,15.153,151.837
C05155=1100.620,99.752,440.195,176.966,15.153,151.838
C05156=1100.613,99.503,440.214,176.963,15.153,151.839
C05157=1100.609,99.254,440.232,176.960,15.153,151.839
C05158=1100.602,99.005,440.250,176.957,15.153,151.840
C05159=1100.597,98.756,440.268,176.954,15.153,151.840
C05160=1100.591,98.506,440.287,176.952,15.153,151.841
C05161=1100.585,98.257,440.305,176.948,15.152,151.842
C05162=1100.579,98.008,440.323,176.946,15.152,151.842
C05163=1100.574,97.758,440.341,176.943,15.152,151.843
C05164=1100.568,97.509,440.360,176.940,15.152,151.843
C05165=1100.563,97.260,440.377,176.938,15.152,151.844
C05166=1100.557,97.010,440.396,176.934,15.152,151.844
C05167=1100.551,96.762,440.414,176.932,15.152,151.845
C05168=1100.545,96.512,440.432,176.929,15.151,151.846
C05169=1100.540,96.239,440.452,176.925,15.151,151.846
C05170=1100.533,95.966,440.471,176.923,15.151,151.847
C05171=1100.527,95.692,440.492,176.919,15.151,151.848
C05172=1100.521,95.420,440.511,176.916,15.151,151.848
C05173=1100.515,95.170,440.529,176.913,15.151,151.849
C05174=1100.510,94.921,440.547,176.910,15.150,151.849
C05175=1100.504,94.672,440.566,176.908,15.150,151.850
C05176=1100.498,94.423,440.584,176.905,15.150,151.850
C05177=1100.492,94.173,440.601,176.902,15.150,151.851
C05178=1100.487,93.923,440.620,176.899,15.150,151.852
C05179=1100.482,93.674,440.637,176.896,15.150,151.852
C05180=1100.475,93.425,440.656,176.894,15.150,151.853
C05181=1100.470,93.176,440.673,176.890,15.149,151.853
C05182=1100.465,92.927,440.692,176.888,15.149,151.854
C05183=1100.459,92.677,440.710,176.885,15.149,151.855
C05184=1100.453,92.428,440.727,176.882,15.149,151.855
C05185=1100.447,92.178,440.745,176.879,15.149,151.856
C05186=1100.442,91.929,440.763,176.877,15.148,151.856
C05187=1100.436,91.681,440.781,176.873,15.148,151.857
C05188=1100.430,91.431,440.799,176.871,15.148,151.857
C05189=1100.425,91.182,440.817,176.868,15.148,151.858
C05190=1100.419,90.933,440.835,176.865,15.148,151.858
C05191=1100.413,90.683,440.852,176.863,15.148,151.859
C05192=1100.408,90.434,440.870,176.859,15.147,151.860
C05193=1100.402,90.184,440.889,176.857,15.147,151.860
C05194=1100.397,89.935,440.906,176.854,15.147,151.861
C05195=1100.391,89.686,440.924,176.851,15.147,151.861
C05196=1100.385,89.436,440.942,176.848,15.146,151.862
C05197=1100.380,89.187,440.959,176.846,15.146,151.862
C05198=1100.374,88.937,440.977,176.842,15.146,151.863
C05199=1100.368,88.688,440.995,176.840,15.146,151.864
C05200=1100.362,88.439,441.012,176.838,15.146,151.864
C05201=1100.356,88.189,441.030,176.834,15.145,151.865
C05202=1100.351,87.940,441.048,176.832,15.145,151.865
C05203=1100.345,87.691,441.065,176.829,15.145,151.866
C05204=1100.339,87.442,441.083,176.826,15.145,151.866
C05205=1100.334,87.193,441.101,176.823,15.144,151.867
C05206=1100.328,86.943,441.119,176.821,15.144,151.867
C05207=1100.322,86.694,441.136,176.818,15.144,151.868
C05208=1100.317,86.445,441.154,176.815,15.144,151.868
C05209=1100.311,86.196,441.171,176.813,15.144,151.869
C05210=1100.305,85.946,441.189,176.809,15.143,151.869
C05211=1100.299,85.697,441.207,176.807,15.143,151.870
C05212=1100.294,85.448,441.225,176.804,15.143,151.871
C05213=1100.288,85.198,441.242,176.802,15.143,151.871
C05214=1100.283,84.949,441.259,176.798,15.142,151.872
C05215=1100.277,84.700,441.277,176.796,15.142,151.872
C05216=1100.271,84.450,441.295,176.794,15.142,151.873
C05217=1100.265,84.201,441.312,176.790,15.141,151.873
C05218=1100.260,83.952,441.330,176.788,15.142,151.874
C05219=1100.254,83.703,441.347,176.785,15.141,151.874
C05220=1100.248,83.452,441.365,176.782,15.141,151.875
C05221=1100.242,83.204,441.382,176.779,15.140,151.875
C05222=1100.237,82.955,441.399,176.777,15.140,151.876
C05223=1100.231,82.705,441.417,176.774,15.140,151.876
C05224=1100.225,82.456,441.435,176.771,15.140,151.877
C05225=1100.220,82.206,441.452,176.769,15.139,151.877
C05226=1100.214,81.957,441.469,176.766,15.139,151.878
C05227=1100.209,81.708,441.487,176.763,15.139,151.878
C05228=1100.203,81.458,441.505,176.760,15.138,151.879
C05229=1100.197,81.209,441.522,176.758,15.138,151.880
C05230=1100.192,80.960,441.539,176.755,15.137,151.880
C05231=1100.186,80.711,441.557,176.752,15.138,151.881
C05232=1100.181,80.461,441.574,176.750,15.137,151.881
C05233=1100.175,80.188,441.592,176.747,15.137,151.882
C05234=1100.168,79.914,441.612,176.743,15.136,151.882
C05235=1100.161,79.642,441.631,176.741,15.136,151.883
C05236=1100.155,79.368,441.650,176.738,15.136,151.883
C05237=1100.150,79.119,441.666,176.735,15.135,151.884
C05238=1100.145,78.870,441.684,176.733,15.135,151.884
C05239=1100.139,78.621,441.702,176.730,15.135,151.885
C05240=1100.134,78.371,441.718,176.727,15.134,151.885
C05241=1100.127,78.122,441.736,176.725,15.134,151.886
C05242=1100.122,77.872,441.753,176.721,15.134,151.886
C05243=1100.116,77.623,441.770,176.719,15.133,151.887
C05244=1100.111,77.374,441.788,176.717,15.134,151.887
C05245=1100.105,77.125,441.804,176.714,15.133,151.888
C05246=1100.099,76.875,441.822,176.711,15.133,151.888
C05247=1100.093,76.625,441.839,176.708,15.132,151.889
C05248=1100.088,76.376,441.856,176.706,15.132,151.889
C05249=1100.082,76.127,441.873,176.703,15.131,151.890
C05250=1100.076,75.878,441.890,176.700,15.131,151.890
C05251=1100.071,75.629,441.908,176.698,15.131,151.891
C05252=1100.064,75.379,441.924,176.695,15.130,151.891
C05253=1100.059,75.130,441.942,176.693,15.130,151.892
C05254=1100.054,74.880,441.959,176.690,15.129,151.892
C05255=1100.047,74.631,441.976,176.687,15.129,151.893
C05256=1100.042,74.382,441.993,176.685,15.129,151.893
C05257=1100.037,74.132,442.010,176.682,15.129,151.894
C05258=1100.031,73.883,442.026,176.680,15.128,151.894
C05259=1100.025,73.633,442.044,176.676,15.128,151.895
C05260=1100.019,73.384,442.061,176.674,15.128,151.895
C05261=1100.013,73.134,442.078,176.671,15.127,151.896
C05262=1100.008,72.885,442.095,176.669,15.127,151.896
C05263=1100.003,72.636,442.112,176.666,15.127,151.897
C05264=1099.996,72.387,442.129,176.663,15.126,151.897
C05265=1099.991,72.137,442.146,176.661,15.126,151.898
C05266=1099.985,71.888,442.162,176.658,15.125,151.898
C05267=1099.980,71.639,442.180,176.655,15.125,151.899
C05268=1099.975,71.389,442.196,176.653,15.125,151.899
C05269=1099.968,71.140,442.214,176.650,15.124,151.900
C05270=1099.962,70.890,442.231,176.648,15.124,151.900
C05271=1099.956,70.641,442.247,176.645,15.123,151.901
C05272=1099.951,70.392,442.264,176.643,15.123,151.901
C05273=1099.946,70.142,442.281,176.640,15.123,151.902
C05274=1099.940,69.893,442.298,176.637,15.122,151.902
C05275=1099.934,69.644,442.315,176.635,15.122,151.902
C05276=1099.928,69.394,442.331,176.632,15.121,151.903
C05277=1099.923,69.145,442.348,176.630,15.121,151.903
C05278=1099.917,68.895,442.364,176.627,15.121,151.904
C05279=1099.912,68.646,442.382,176.624,15.120,151.904
C05280=1099.906,68.397,442.398,176.622,15.120,151.905
C05281=1099.900,68.147,442.415,176.619,15.119,151.905
C05282=1099.895,67.898,442.431,176.617,15.119,151.906
C05283=1099.889,67.649,442.449,176.615,15.118,151.906
C05284=1099.883,67.400,442.465,176.611,15.118,151.907
C05285=1099.878,67.150,442.482,176.609,15.118,151.907
C05286=1099.871,66.900,442.499,176.606,15.117,151.908
C05287=1099.865,66.651,442.516,176.604,15.117,151.908
C05288=1099.860,66.401,442.533,176.601,15.117,151.909
C05289=1099.854,66.152,442.549,176.599,15.116,151.909
C05290=1099.849,65.902,442.566,176.596,15.115,151.909
C05291=1099.843,65.653,442.582,176.593,15.114,151.910
C05292=1099.837,65.404,442.599,176.591,15.115,151.910
C05293=1099.831,65.155,442.616,176.589,15.114,151.911
C05294=1099.825,64.905,442.632,176.586,15.113,151.911
C05295=1099.820,64.656,442.649,176.584,15.113,151.912
C05296=1099.814,64.406,442.665,176.581,15.113,151.912
C05297=1099.808,64.133,442.684,176.578,15.112,151.913
C05298=1099.802,63.860,442.701,176.575,15.111,151.913
C05299=1099.796,63.587,442.719,176.573,15.112,151.914
C05300=1099.789,63.314,442.737,176.570,15.111,151.914
C05301=1099.784,63.064,442.754,176.567,15.111,151.915
C05302=1099.778,62.815,442.770,176.564,15.110,151.915
C05303=1099.772,62.566,442.787,176.562,15.110,151.916
C05304=1099.766,62.316,442.803,176.560,15.109,151.916
C05305=1099.761,62.067,442.820,176.557,15.108,151.916
C05306=1099.755,61.817,442.836,176.554,15.109,151.917
C05307=1099.749,61.568,442.852,176.552,15.108,151.917
C05308=1099.743,61.319,442.868,176.549,15.107,151.918
C05309=1099.737,61.069,442.885,176.547,15.107,151.918
C05310=1099.732,60.820,442.902,176.544,15.106,151.919
C05311=1099.726,60.570,442.918,176.542,15.106,151.919
C05312=1099.720,60.321,442.934,176.539,15.106,151.920
C05313=1099.714,60.072,442.950,176.536,15.105,151.920
C05314=1099.708,59.822,442.967,176.534,15.105,151.921
C05315=1099.702,59.573,442.983,176.532,15.105,151.921
C05316=1099.697,59.323,443.000,176.529,15.104,151.921
C05317=1099.691,59.074,443.016,176.527,15.103,151.922
C05318=1099.685,58.825,443.032,176.524,15.102,151.922
C05319=1099.679,58.575,443.049,176.522,15.102,151.923
C05320=1099.673,58.326,443.065,176.520,15.102,151.923
C05321=1099.668,58.076,443.082,176.516,15.101,151.924
C05322=1099.662,57.827,443.098,176.514,15.101,151.924
C05323=1099.656,57.578,443.114,176.512,15.101,151.925
C05324=1099.650,57.328,443.130,176.509,15.100,151.925
C05325=1099.645,57.079,443.147,176.507,15.100,151.925
C05326=1099.639,56.829,443.162,176.505,15.099,151.926
C05327=1099.633,56.580,443.179,176.502,15.098,151.926
C05328=1099.628,56.331,443.195,176.499,15.098,151.927
C05329=1099.622,56.081,443.211,176.496,15.097,151.927
C05330=1099.616,55.832,443.227,176.494,15.097,151.928
C05331=1099.610,55.583,443.244,176.492,15.097,151.928
C05332=1099.605,55.332,443.260,176.489,15.096,151.928
C05333=1099.599,55.084,443.276,176.487,15.095,151.929
C05334=1099.593,54.834,443.292,176.485,15.095,151.929
C05335=1099.587,54.585,443.308,176.482,15.094,151.930
C05336=1099.582,54.336,443.324,176.480,15.094,151.930
C05337=1099.576,54.086,443.340,176.477,15.094,151.930
C05338=1099.570,53.836,443.356,176.474,15.093,151.931
C05339=1099.564,53.587,443.372,176.472,15.092,151.931
C05340=1099.559,53.338,443.388,176.470,15.092,151.932
C05341=1099.553,53.088,443.404,176.467,15.091,151.932
C05342=1099.548,52.839,443.421,176.465,15.090,151.932
C05343=1099.542,52.589,443.437,176.462,15.090,151.933
C05344=1099.536,52.339,443.453,176.460,15.089,151.933
C05345=1099.531,52.091,443.468,176.458,15.089,151.934
C05346=1099.525,51.841,443.485,176.455,15.088,151.934
C05347=1099.519,51.591,443.500,176.453,15.088,151.935
C05348=1099.513,51.342,443.516,176.450,15.087,151.935
C05349=1099.507,51.093,443.533,176.448,15.087,151.935
C05350=1099.502,50.843,443.548,176.445,15.086,151.936
C05351=1099.496,50.594,443.564,176.443,15.085,151.936
C05352=1099.490,50.345,443.580,176.441,15.085,151.937
C05353=1099.485,50.095,443.596,176.438,15.084,151.937
C05354=1099.479,49.846,443.612,176.436,15.084,151.937
C05355=1099.473,49.597,443.628,176.433,15.083,151.938
C05356=1099.468,49.347,443.644,176.431,15.083,151.938
C05357=1099.462,49.097,443.660,176.429,15.082,151.938
C05358=1099.457,48.848,443.675,176.426,15.081,151.939
C05359=1099.451,48.599,443.691,176.424,15.081,151.939
C05360=1099.445,48.349,443.707,176.422,15.081,151.940
C05361=1099.439,48.075,443.724,176.419,15.080,151.940
C05362=1099.434,47.802,443.742,176.416,15.079,151.941
C05363=1099.427,47.529,443.760,176.414,15.078,151.941
C05364=1099.421,47.255,443.777,176.411,15.078,151.941
C05365=1099.415,47.006,443.793,176.409,15.077,151.942
C05366=1099.410,46.756,443.808,176.407,15.077,151.942
C05367=1099.404,46.507,443.824,176.404,15.076,151.943
C05368=1099.398,46.257,443.840,176.401,15.075,151.943
C05369=1099.393,46.008,443.856,176.400,15.075,151.943
C05370=1099.387,45.758,443.871,176.397,15.074,151.944
C05371=1099.381,45.509,443.888,176.394,15.073,151.944
C05372=1099.375,45.260,443.902,176.392,15.073,151.945
C05373=1099.370,45.011,443.919,176.390,15.072,151.945
C05374=1099.364,44.761,443.934,176.387,15.071,151.945
C05375=1099.359,44.512,443.950,176.385,15.071,151.946
C05376=1099.353,44.262,443.966,176.383,15.070,151.946
C05377=1099.348,44.013,443.981,176.380,15.069,151.946
C05378=1099.342,43.763,443.997,176.378,15.069,151.947
C05379=1099.336,43.513,444.012,176.375,15.068,151.947
C05380=1099.330,43.264,444.029,176.373,15.068,151.947
C05381=1099.325,43.015,444.044,176.371,15.067,151.948
C05382=1099.319,42.765,444.059,176.368,15.066,151.948
C05383=1099.313,42.516,444.075,176.366,15.066,151.949
C05384=1099.308,42.266,444.090,176.364,15.065,151.949
C05385=1099.302,42.017,444.106,176.361,15.064,151.949
C05386=1099.296,41.767,444.122,176.359,15.064,151.950
C05387=1099.291,41.518,444.137,176.357,15.063,151.950
C05388=1099.285,41.268,444.152,176.354,15.062,151.951
C05389=1099.279,41.019,444.168,176.352,15.062,151.951
C05390=1099.274,40.770,444.184,176.350,15.061,151.951
C05391=1099.267,40.520,444.199,176.347,15.061,151.952
C05392=1099.262,40.271,444.214,176.345,15.060,151.952
C05393=1099.256,40.021,444.230,176.343,15.059,151.952
C05394=1099.251,39.771,444.246,176.340,15.059,151.953
C05395=1099.245,39.522,444.260,176.338,15.058,151.953
C05396=1099.239,39.273,444.276,176.336,15.058,151.953
C05397=1099.233,39.023,444.292,176.333,15.057,151.954
C05398=1099.228,38.774,444.307,176.331,15.056,151.954
C05399=1099.222,38.524,444.322,176.329,15.056,151.955
C05400=1099.217,38.276,444.338,176.327,15.055,151.955
C05401=1099.211,38.026,444.353,176.324,15.054,151.955
C05402=1099.205,37.776,444.368,176.322,15.054,151.956
C05403=1099.200,37.527,444.384,176.320,15.053,151.956
C05404=1099.194,37.277,444.400,176.317,15.052,151.956
C05405=1099.187,37.028,444.415,176.315,15.052,151.957
C05406=1099.182,36.778,444.430,176.313,15.051,151.957
C05407=1099.176,36.529,444.445,176.310,15.050,151.957
C05408=1099.171,36.279,444.460,176.308,15.050,151.958
C05409=1099.165,36.029,444.476,176.306,15.050,151.958
C05410=1099.158,35.780,444.491,176.304,15.049,151.959
C05411=1099.153,35.531,444.506,176.301,15.048,151.959
C05412=1099.147,35.282,444.521,176.299,15.047,151.959
C05413=1099.142,35.032,444.537,176.297,15.047,151.960
C05414=1099.136,34.783,444.552,176.294,15.046,151.960
C05415=1099.130,34.533,444.567,176.292,15.045,151.960
C05416=1099.125,34.283,444.582,176.290,15.045,151.961
C05417=1099.119,34.034,444.597,176.287,15.044,151.961
C05418=1099.113,33.785,444.613,176.285,15.043,151.961
C05419=1099.107,33.535,444.628,176.283,15.043,151.962
C05420=1099.102,33.286,444.643,176.281,15.042,151.962
C05421=1099.095,33.036,444.658,176.278,15.041,151.963
C05422=1099.090,32.787,444.673,176.276,15.041,151.963
C05423=1099.084,32.538,444.688,176.274,15.040,151.963
C05424=1099.078,32.288,444.704,176.271,15.039,151.964
C05425=1099.072,32.015,444.720,176.269,15.039,151.964
C05426=1099.066,31.741,444.736,176.266,15.038,151.964
C05427=1099.060,31.467,444.753,176.264,15.037,151.965
C05428=1099.054,31.195,444.770,176.261,15.036,151.965
C05429=1099.048,30.945,444.785,176.259,15.035,151.965
C05430=1099.042,30.696,444.800,176.257,15.035,151.966
C05431=1099.037,30.445,444.815,176.255,15.034,151.966
C05432=1099.031,30.196,444.829,176.252,15.033,151.966
C05433=1099.025,29.946,444.845,176.250,15.033,151.967
C05434=1099.020,29.697,444.859,176.248,15.032,151.967
C05435=1099.014,29.447,444.875,176.246,15.032,151.967
C05436=1099.008,29.198,444.890,176.243,15.031,151.968
C05437=1099.002,28.949,444.905,176.241,15.030,151.968
C05438=1098.997,28.699,444.920,176.239,15.030,151.969
C05439=1098.990,28.450,444.935,176.237,15.028,151.969
C05440=1098.985,28.200,444.950,176.234,15.028,151.969
C05441=1098.979,27.951,444.965,176.233,15.027,151.969
C05442=1098.973,27.702,444.979,176.230,15.027,151.970
